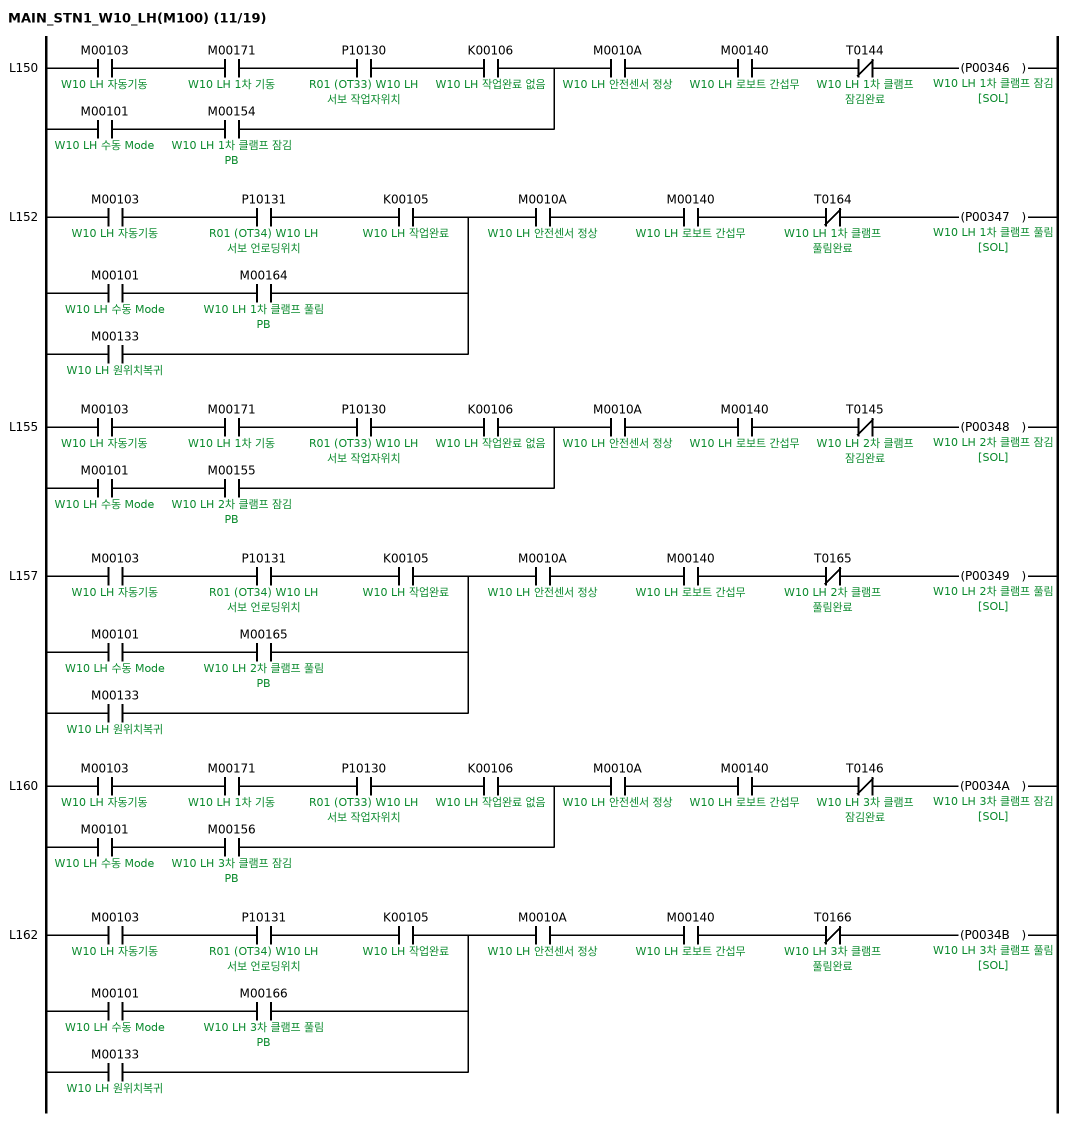
[picture p48: MAIN_STN1_W10_LH(M100) rungs L150-L162]
; L150
LOAD      M00103	// W10 LH 자동기동
AND       M00171	// W10 LH 1차 기동
AND       P10130	// R01 (OT33) W10 LH 서보 작업자위치
AND       K00106	// W10 LH 작업완료 없음
LOAD      M00101	// W10 LH 수동 Mode
AND       M00154	// W10 LH 1차 클램프 잠김 PB
OR LOAD
AND       M0010A	// W10 LH 안전센서 정상
AND       M00140	// W10 LH 로보트 간섭무
AND NOT   T0144	// W10 LH 1차 클램프 잠김완료
OUT       P00346	// W10 LH 1차 클램프 잠김 [SOL]
; L152
LOAD      M00103	// W10 LH 자동기동
AND       P10131	// R01 (OT34) W10 LH 서보 언로딩위치
AND       K00105	// W10 LH 작업완료
LOAD      M00101	// W10 LH 수동 Mode
AND       M00164	// W10 LH 1차 클램프 풀림 PB
OR LOAD
OR        M00133	// W10 LH 원위치복귀
AND       M0010A	// W10 LH 안전센서 정상
AND       M00140	// W10 LH 로보트 간섭무
AND NOT   T0164	// W10 LH 1차 클램프 풀림완료
OUT       P00347	// W10 LH 1차 클램프 풀림 [SOL]
; L155
LOAD      M00103	// W10 LH 자동기동
AND       M00171	// W10 LH 1차 기동
AND       P10130	// R01 (OT33) W10 LH 서보 작업자위치
AND       K00106	// W10 LH 작업완료 없음
LOAD      M00101	// W10 LH 수동 Mode
AND       M00155	// W10 LH 2차 클램프 잠김 PB
OR LOAD
AND       M0010A	// W10 LH 안전센서 정상
AND       M00140	// W10 LH 로보트 간섭무
AND NOT   T0145	// W10 LH 2차 클램프 잠김완료
OUT       P00348	// W10 LH 2차 클램프 잠김 [SOL]
; L157
LOAD      M00103	// W10 LH 자동기동
AND       P10131	// R01 (OT34) W10 LH 서보 언로딩위치
AND       K00105	// W10 LH 작업완료
LOAD      M00101	// W10 LH 수동 Mode
AND       M00165	// W10 LH 2차 클램프 풀림 PB
OR LOAD
OR        M00133	// W10 LH 원위치복귀
AND       M0010A	// W10 LH 안전센서 정상
AND       M00140	// W10 LH 로보트 간섭무
AND NOT   T0165	// W10 LH 2차 클램프 풀림완료
OUT       P00349	// W10 LH 2차 클램프 풀림 [SOL]
; L160
LOAD      M00103	// W10 LH 자동기동
AND       M00171	// W10 LH 1차 기동
AND       P10130	// R01 (OT33) W10 LH 서보 작업자위치
AND       K00106	// W10 LH 작업완료 없음
LOAD      M00101	// W10 LH 수동 Mode
AND       M00156	// W10 LH 3차 클램프 잠김 PB
OR LOAD
AND       M0010A	// W10 LH 안전센서 정상
AND       M00140	// W10 LH 로보트 간섭무
AND NOT   T0146	// W10 LH 3차 클램프 잠김완료
OUT       P0034A	// W10 LH 3차 클램프 잠김 [SOL]
; L162
LOAD      M00103	// W10 LH 자동기동
AND       P10131	// R01 (OT34) W10 LH 서보 언로딩위치
AND       K00105	// W10 LH 작업완료
LOAD      M00101	// W10 LH 수동 Mode
AND       M00166	// W10 LH 3차 클램프 풀림 PB
OR LOAD
OR        M00133	// W10 LH 원위치복귀
AND       M0010A	// W10 LH 안전센서 정상
AND       M00140	// W10 LH 로보트 간섭무
AND NOT   T0166	// W10 LH 3차 클램프 풀림완료
OUT       P0034B	// W10 LH 3차 클램프 풀림 [SOL]

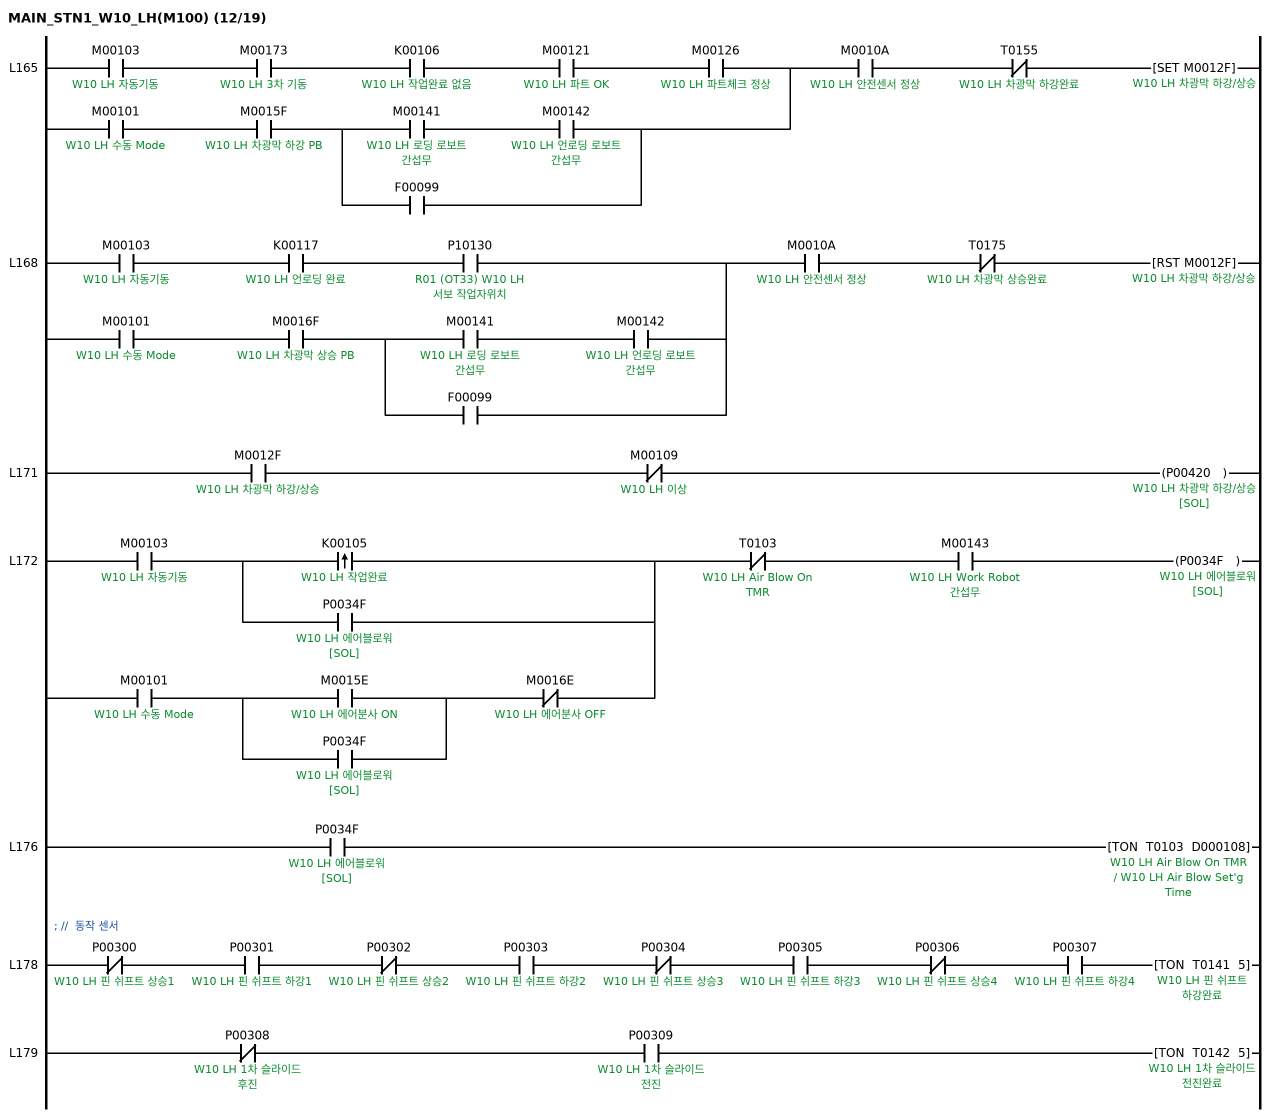
; L165
LOAD      M00103	// W10 LH 자동기동
AND       M00173	// W10 LH 3차 기동
AND       K00106	// W10 LH 작업완료 없음
AND       M00121	// W10 LH 파트 OK
AND       M00126	// W10 LH 파트체크 정상
LOAD      M00101	// W10 LH 수동 Mode
AND       M0015F	// W10 LH 차광막 하강 PB
LOAD      M00141	// W10 LH 로딩 로보트 간섭무
AND       M00142	// W10 LH 언로딩 로보트 간섭무
OR        F00099
AND LOAD
OR LOAD
AND       M0010A	// W10 LH 안전센서 정상
AND NOT   T0155	// W10 LH 차광막 하강완료
SET       M0012F	// W10 LH 차광막 하강/상승
; L168
LOAD      M00103	// W10 LH 자동기동
AND       K00117	// W10 LH 언로딩 완료
AND       P10130	// R01 (OT33) W10 LH 서보 작업자위치
LOAD      M00101	// W10 LH 수동 Mode
AND       M0016F	// W10 LH 차광막 상승 PB
LOAD      M00141	// W10 LH 로딩 로보트 간섭무
AND       M00142	// W10 LH 언로딩 로보트 간섭무
OR        F00099
AND LOAD
OR LOAD
AND       M0010A	// W10 LH 안전센서 정상
AND NOT   T0175	// W10 LH 차광막 상승완료
RST       M0012F	// W10 LH 차광막 하강/상승
; L171
LOAD      M0012F	// W10 LH 차광막 하강/상승
AND NOT   M00109	// W10 LH 이상
OUT       P00420	// W10 LH 차광막 하강/상승 [SOL]
; L172
LOAD      M00103	// W10 LH 자동기동
LOADP     K00105	// W10 LH 작업완료
OR        P0034F	// W10 LH 에어블로워 [SOL]
AND LOAD
LOAD      M00101	// W10 LH 수동 Mode
LOAD      M0015E	// W10 LH 에어분사 ON
OR        P0034F	// W10 LH 에어블로워 [SOL]
AND LOAD
AND NOT   M0016E	// W10 LH 에어분사 OFF
OR LOAD
AND NOT   T0103	// W10 LH Air Blow On TMR
AND       M00143	// W10 LH Work Robot 간섭무
OUT       P0034F	// W10 LH 에어블로워 [SOL]
; L176
LOAD      P0034F	// W10 LH 에어블로워 [SOL]
TON       T0103 D000108	// W10 LH Air Blow On TMR / W10 LH Air Blow Set'g Time
//   //  동작 센서
; L178
LOAD NOT  P00300	// W10 LH 핀 쉬프트 상승1
AND       P00301	// W10 LH 핀 쉬프트 하강1
AND NOT   P00302	// W10 LH 핀 쉬프트 상승2
AND       P00303	// W10 LH 핀 쉬프트 하강2
AND NOT   P00304	// W10 LH 핀 쉬프트 상승3
AND       P00305	// W10 LH 핀 쉬프트 하강3
AND NOT   P00306	// W10 LH 핀 쉬프트 상승4
AND       P00307	// W10 LH 핀 쉬프트 하강4
TON       T0141 5	// W10 LH 핀 쉬프트 하강완료
; L179
LOAD NOT  P00308	// W10 LH 1차 슬라이드 후진
AND       P00309	// W10 LH 1차 슬라이드 전진
TON       T0142 5	// W10 LH 1차 슬라이드 전진완료

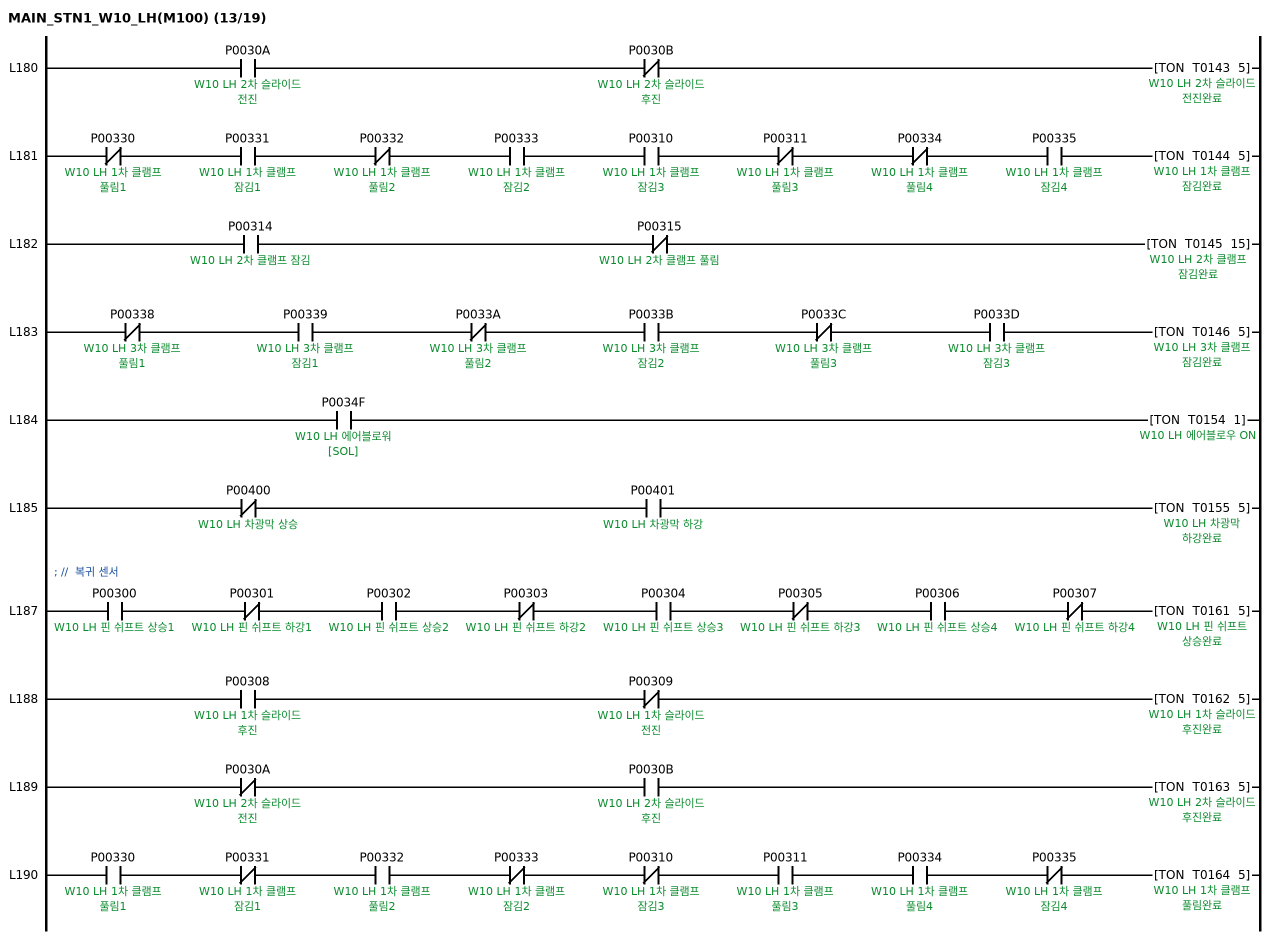
; L180
LOAD      P0030A	// W10 LH 2차 슬라이드 전진
AND NOT   P0030B	// W10 LH 2차 슬라이드 후진
TON       T0143 5	// W10 LH 2차 슬라이드 전진완료
; L181
LOAD NOT  P00330	// W10 LH 1차 클램프 풀림1
AND       P00331	// W10 LH 1차 클램프 잠김1
AND NOT   P00332	// W10 LH 1차 클램프 풀림2
AND       P00333	// W10 LH 1차 클램프 잠김2
AND       P00310	// W10 LH 1차 클램프 잠김3
AND NOT   P00311	// W10 LH 1차 클램프 풀림3
AND NOT   P00334	// W10 LH 1차 클램프 풀림4
AND       P00335	// W10 LH 1차 클램프 잠김4
TON       T0144 5	// W10 LH 1차 클램프 잠김완료
; L182
LOAD      P00314	// W10 LH 2차 클램프 잠김
AND NOT   P00315	// W10 LH 2차 클램프 풀림
TON       T0145 15	// W10 LH 2차 클램프 잠김완료
; L183
LOAD NOT  P00338	// W10 LH 3차 클램프 풀림1
AND       P00339	// W10 LH 3차 클램프 잠김1
AND NOT   P0033A	// W10 LH 3차 클램프 풀림2
AND       P0033B	// W10 LH 3차 클램프 잠김2
AND NOT   P0033C	// W10 LH 3차 클램프 풀림3
AND       P0033D	// W10 LH 3차 클램프 잠김3
TON       T0146 5	// W10 LH 3차 클램프 잠김완료
; L184
LOAD      P0034F	// W10 LH 에어블로워 [SOL]
TON       T0154 1	// W10 LH 에어블로우 ON
; L185
LOAD NOT  P00400	// W10 LH 차광막 상승
AND       P00401	// W10 LH 차광막 하강
TON       T0155 5	// W10 LH 차광막 하강완료
//   //  복귀 센서
; L187
LOAD      P00300	// W10 LH 핀 쉬프트 상승1
AND NOT   P00301	// W10 LH 핀 쉬프트 하강1
AND       P00302	// W10 LH 핀 쉬프트 상승2
AND NOT   P00303	// W10 LH 핀 쉬프트 하강2
AND       P00304	// W10 LH 핀 쉬프트 상승3
AND NOT   P00305	// W10 LH 핀 쉬프트 하강3
AND       P00306	// W10 LH 핀 쉬프트 상승4
AND NOT   P00307	// W10 LH 핀 쉬프트 하강4
TON       T0161 5	// W10 LH 핀 쉬프트 상승완료
; L188
LOAD      P00308	// W10 LH 1차 슬라이드 후진
AND NOT   P00309	// W10 LH 1차 슬라이드 전진
TON       T0162 5	// W10 LH 1차 슬라이드 후진완료
; L189
LOAD NOT  P0030A	// W10 LH 2차 슬라이드 전진
AND       P0030B	// W10 LH 2차 슬라이드 후진
TON       T0163 5	// W10 LH 2차 슬라이드 후진완료
; L190
LOAD      P00330	// W10 LH 1차 클램프 풀림1
AND NOT   P00331	// W10 LH 1차 클램프 잠김1
AND       P00332	// W10 LH 1차 클램프 풀림2
AND NOT   P00333	// W10 LH 1차 클램프 잠김2
AND NOT   P00310	// W10 LH 1차 클램프 잠김3
AND       P00311	// W10 LH 1차 클램프 풀림3
AND       P00334	// W10 LH 1차 클램프 풀림4
AND NOT   P00335	// W10 LH 1차 클램프 잠김4
TON       T0164 5	// W10 LH 1차 클램프 풀림완료

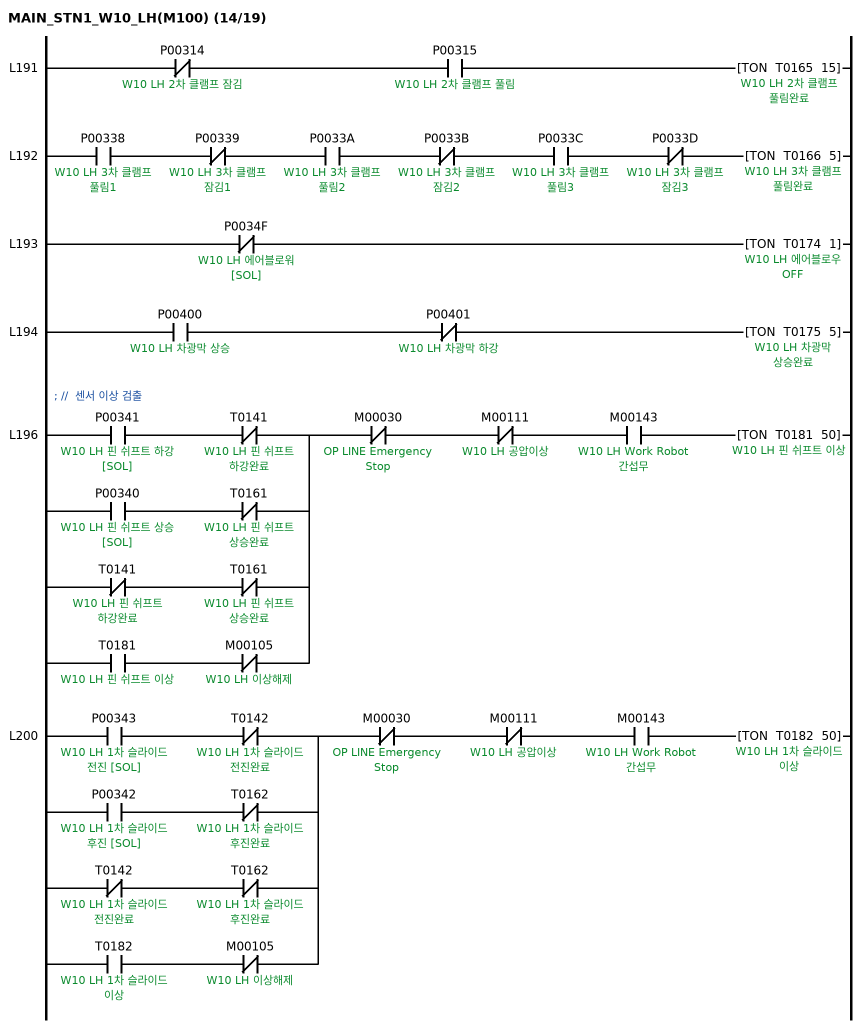
; L191
LOAD NOT  P00314	// W10 LH 2차 클램프 잠김
AND       P00315	// W10 LH 2차 클램프 풀림
TON       T0165 15	// W10 LH 2차 클램프 풀림완료
; L192
LOAD      P00338	// W10 LH 3차 클램프 풀림1
AND NOT   P00339	// W10 LH 3차 클램프 잠김1
AND       P0033A	// W10 LH 3차 클램프 풀림2
AND NOT   P0033B	// W10 LH 3차 클램프 잠김2
AND       P0033C	// W10 LH 3차 클램프 풀림3
AND NOT   P0033D	// W10 LH 3차 클램프 잠김3
TON       T0166 5	// W10 LH 3차 클램프 풀림완료
; L193
LOAD NOT  P0034F	// W10 LH 에어블로워 [SOL]
TON       T0174 1	// W10 LH 에어블로우 OFF
; L194
LOAD      P00400	// W10 LH 차광막 상승
AND NOT   P00401	// W10 LH 차광막 하강
TON       T0175 5	// W10 LH 차광막 상승완료
//     //  센서 이상 검출
; L196
LOAD      P00341	// W10 LH 핀 쉬프트 하강 [SOL]
AND NOT   T0141	// W10 LH 핀 쉬프트 하강완료
LOAD      P00340	// W10 LH 핀 쉬프트 상승 [SOL]
AND NOT   T0161	// W10 LH 핀 쉬프트 상승완료
OR LOAD
LOAD NOT  T0141	// W10 LH 핀 쉬프트 하강완료
AND NOT   T0161	// W10 LH 핀 쉬프트 상승완료
OR LOAD
LOAD      T0181	// W10 LH 핀 쉬프트 이상
AND NOT   M00105	// W10 LH 이상해제
OR LOAD
AND NOT   M00030	// OP LINE Emergency Stop
AND NOT   M00111	// W10 LH 공압이상
AND       M00143	// W10 LH Work Robot 간섭무
TON       T0181 50	// W10 LH 핀 쉬프트 이상
; L200
LOAD      P00343	// W10 LH 1차 슬라이드 전진 [SOL]
AND NOT   T0142	// W10 LH 1차 슬라이드 전진완료
LOAD      P00342	// W10 LH 1차 슬라이드 후진 [SOL]
AND NOT   T0162	// W10 LH 1차 슬라이드 후진완료
OR LOAD
LOAD NOT  T0142	// W10 LH 1차 슬라이드 전진완료
AND NOT   T0162	// W10 LH 1차 슬라이드 후진완료
OR LOAD
LOAD      T0182	// W10 LH 1차 슬라이드 이상
AND NOT   M00105	// W10 LH 이상해제
OR LOAD
AND NOT   M00030	// OP LINE Emergency Stop
AND NOT   M00111	// W10 LH 공압이상
AND       M00143	// W10 LH Work Robot 간섭무
TON       T0182 50	// W10 LH 1차 슬라이드 이상

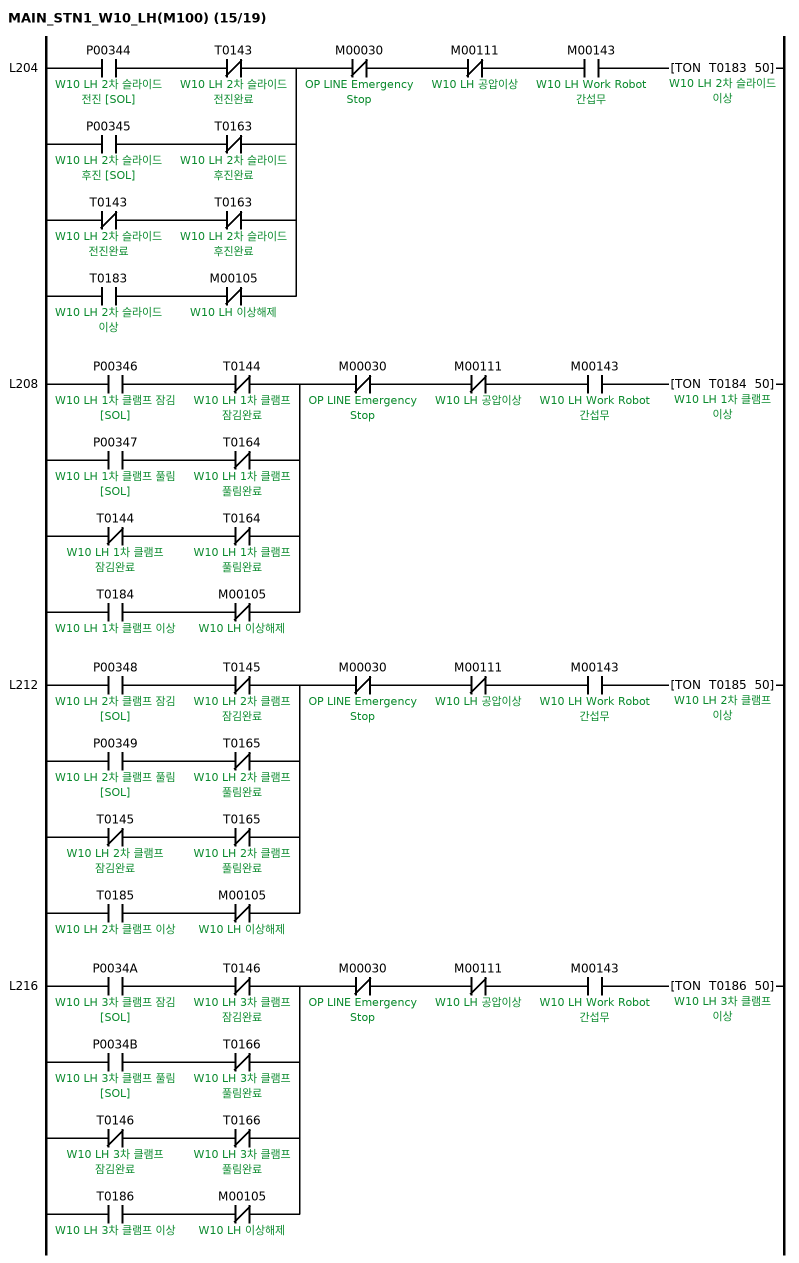
; L204
LOAD      P00344	// W10 LH 2차 슬라이드 전진 [SOL]
AND NOT   T0143	// W10 LH 2차 슬라이드 전진완료
LOAD      P00345	// W10 LH 2차 슬라이드 후진 [SOL]
AND NOT   T0163	// W10 LH 2차 슬라이드 후진완료
OR LOAD
LOAD NOT  T0143	// W10 LH 2차 슬라이드 전진완료
AND NOT   T0163	// W10 LH 2차 슬라이드 후진완료
OR LOAD
LOAD      T0183	// W10 LH 2차 슬라이드 이상
AND NOT   M00105	// W10 LH 이상해제
OR LOAD
AND NOT   M00030	// OP LINE Emergency Stop
AND NOT   M00111	// W10 LH 공압이상
AND       M00143	// W10 LH Work Robot 간섭무
TON       T0183 50	// W10 LH 2차 슬라이드 이상
; L208
LOAD      P00346	// W10 LH 1차 클램프 잠김 [SOL]
AND NOT   T0144	// W10 LH 1차 클램프 잠김완료
LOAD      P00347	// W10 LH 1차 클램프 풀림 [SOL]
AND NOT   T0164	// W10 LH 1차 클램프 풀림완료
OR LOAD
LOAD NOT  T0144	// W10 LH 1차 클램프 잠김완료
AND NOT   T0164	// W10 LH 1차 클램프 풀림완료
OR LOAD
LOAD      T0184	// W10 LH 1차 클램프 이상
AND NOT   M00105	// W10 LH 이상해제
OR LOAD
AND NOT   M00030	// OP LINE Emergency Stop
AND NOT   M00111	// W10 LH 공압이상
AND       M00143	// W10 LH Work Robot 간섭무
TON       T0184 50	// W10 LH 1차 클램프 이상
; L212
LOAD      P00348	// W10 LH 2차 클램프 잠김 [SOL]
AND NOT   T0145	// W10 LH 2차 클램프 잠김완료
LOAD      P00349	// W10 LH 2차 클램프 풀림 [SOL]
AND NOT   T0165	// W10 LH 2차 클램프 풀림완료
OR LOAD
LOAD NOT  T0145	// W10 LH 2차 클램프 잠김완료
AND NOT   T0165	// W10 LH 2차 클램프 풀림완료
OR LOAD
LOAD      T0185	// W10 LH 2차 클램프 이상
AND NOT   M00105	// W10 LH 이상해제
OR LOAD
AND NOT   M00030	// OP LINE Emergency Stop
AND NOT   M00111	// W10 LH 공압이상
AND       M00143	// W10 LH Work Robot 간섭무
TON       T0185 50	// W10 LH 2차 클램프 이상
; L216
LOAD      P0034A	// W10 LH 3차 클램프 잠김 [SOL]
AND NOT   T0146	// W10 LH 3차 클램프 잠김완료
LOAD      P0034B	// W10 LH 3차 클램프 풀림 [SOL]
AND NOT   T0166	// W10 LH 3차 클램프 풀림완료
OR LOAD
LOAD NOT  T0146	// W10 LH 3차 클램프 잠김완료
AND NOT   T0166	// W10 LH 3차 클램프 풀림완료
OR LOAD
LOAD      T0186	// W10 LH 3차 클램프 이상
AND NOT   M00105	// W10 LH 이상해제
OR LOAD
AND NOT   M00030	// OP LINE Emergency Stop
AND NOT   M00111	// W10 LH 공압이상
AND       M00143	// W10 LH Work Robot 간섭무
TON       T0186 50	// W10 LH 3차 클램프 이상

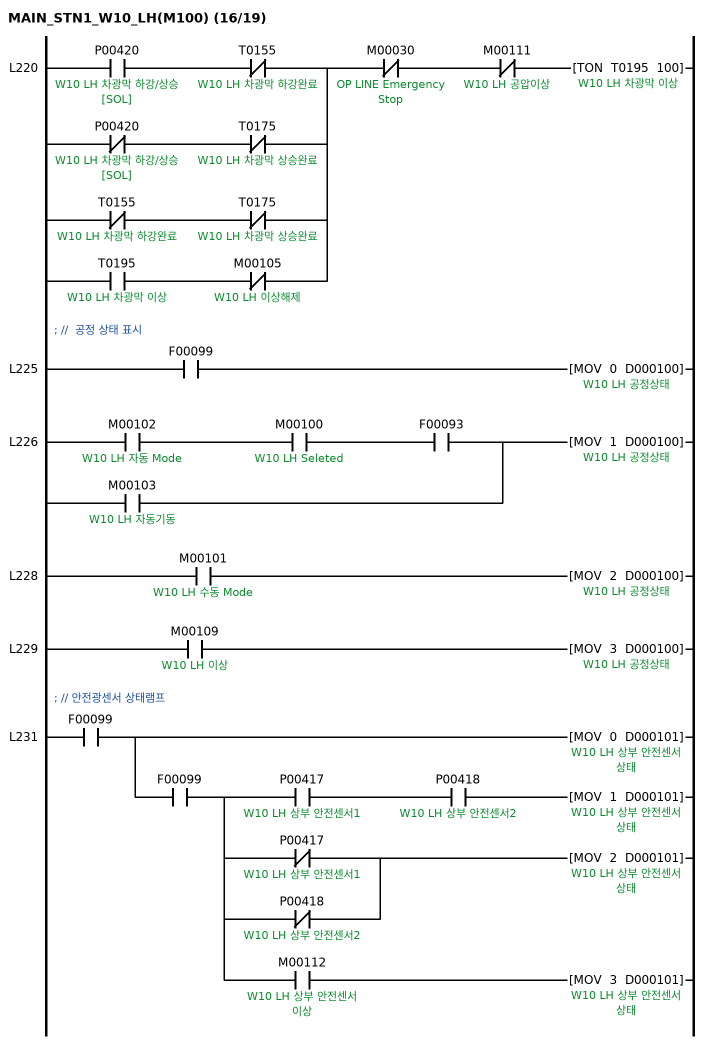
; L220
LOAD      P00420	// W10 LH 차광막 하강/상승 [SOL]
AND NOT   T0155	// W10 LH 차광막 하강완료
LOAD NOT  P00420	// W10 LH 차광막 하강/상승 [SOL]
AND NOT   T0175	// W10 LH 차광막 상승완료
OR LOAD
LOAD NOT  T0155	// W10 LH 차광막 하강완료
AND NOT   T0175	// W10 LH 차광막 상승완료
OR LOAD
LOAD      T0195	// W10 LH 차광막 이상
AND NOT   M00105	// W10 LH 이상해제
OR LOAD
AND NOT   M00030	// OP LINE Emergency Stop
AND NOT   M00111	// W10 LH 공압이상
TON       T0195 100	// W10 LH 차광막 이상
//   //  공정 상태 표시
; L225
LOAD      F00099
MOV       0 D000100	// W10 LH 공정상태
; L226
LOAD      M00102	// W10 LH 자동 Mode
AND       M00100	// W10 LH Seleted
AND       F00093
OR        M00103	// W10 LH 자동기동
MOV       1 D000100	// W10 LH 공정상태
; L228
LOAD      M00101	// W10 LH 수동 Mode
MOV       2 D000100	// W10 LH 공정상태
; L229
LOAD      M00109	// W10 LH 이상
MOV       3 D000100	// W10 LH 공정상태
//   // 안전광센서 상태램프
; L231
LOAD      F00099
MOV       0 D000101	// W10 LH 상부 안전센서 상태
AND       F00099
MPUSH
AND       P00417	// W10 LH 상부 안전센서1
AND       P00418	// W10 LH 상부 안전센서2
MOV       1 D000101	// W10 LH 상부 안전센서 상태
MLOAD
LOAD NOT  P00417	// W10 LH 상부 안전센서1
OR NOT    P00418	// W10 LH 상부 안전센서2
AND LOAD
MOV       2 D000101	// W10 LH 상부 안전센서 상태
MPOP
AND       M00112	// W10 LH 상부 안전센서 이상
MOV       3 D000101	// W10 LH 상부 안전센서 상태

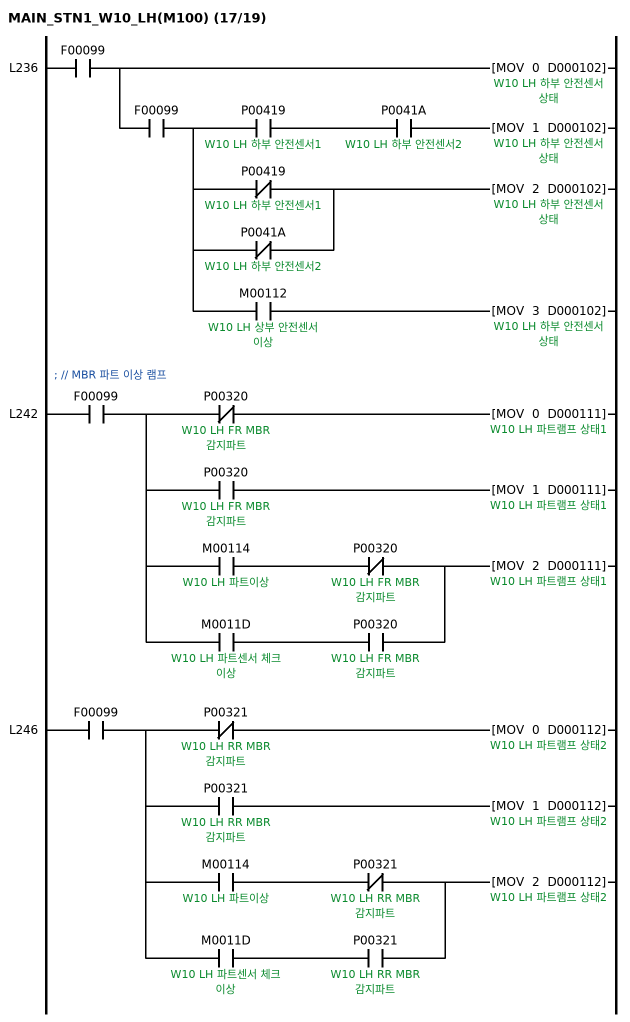
; L236
LOAD      F00099
MOV       0 D000102	// W10 LH 하부 안전센서 상태
AND       F00099
MPUSH
AND       P00419	// W10 LH 하부 안전센서1
AND       P0041A	// W10 LH 하부 안전센서2
MOV       1 D000102	// W10 LH 하부 안전센서 상태
MLOAD
LOAD NOT  P00419	// W10 LH 하부 안전센서1
OR NOT    P0041A	// W10 LH 하부 안전센서2
AND LOAD
MOV       2 D000102	// W10 LH 하부 안전센서 상태
MPOP
AND       M00112	// W10 LH 상부 안전센서 이상
MOV       3 D000102	// W10 LH 하부 안전센서 상태
//   // MBR 파트 이상 램프
; L242
LOAD      F00099
MPUSH
AND NOT   P00320	// W10 LH FR MBR 감지파트
MOV       0 D000111	// W10 LH 파트램프 상태1
MLOAD
AND       P00320	// W10 LH FR MBR 감지파트
MOV       1 D000111	// W10 LH 파트램프 상태1
MPOP
LOAD      M00114	// W10 LH 파트이상
AND NOT   P00320	// W10 LH FR MBR 감지파트
LOAD      M0011D	// W10 LH 파트센서 체크 이상
AND       P00320	// W10 LH FR MBR 감지파트
OR LOAD
AND LOAD
MOV       2 D000111	// W10 LH 파트램프 상태1
; L246
LOAD      F00099
MPUSH
AND NOT   P00321	// W10 LH RR MBR 감지파트
MOV       0 D000112	// W10 LH 파트램프 상태2
MLOAD
AND       P00321	// W10 LH RR MBR 감지파트
MOV       1 D000112	// W10 LH 파트램프 상태2
MPOP
LOAD      M00114	// W10 LH 파트이상
AND NOT   P00321	// W10 LH RR MBR 감지파트
LOAD      M0011D	// W10 LH 파트센서 체크 이상
AND       P00321	// W10 LH RR MBR 감지파트
OR LOAD
AND LOAD
MOV       2 D000112	// W10 LH 파트램프 상태2

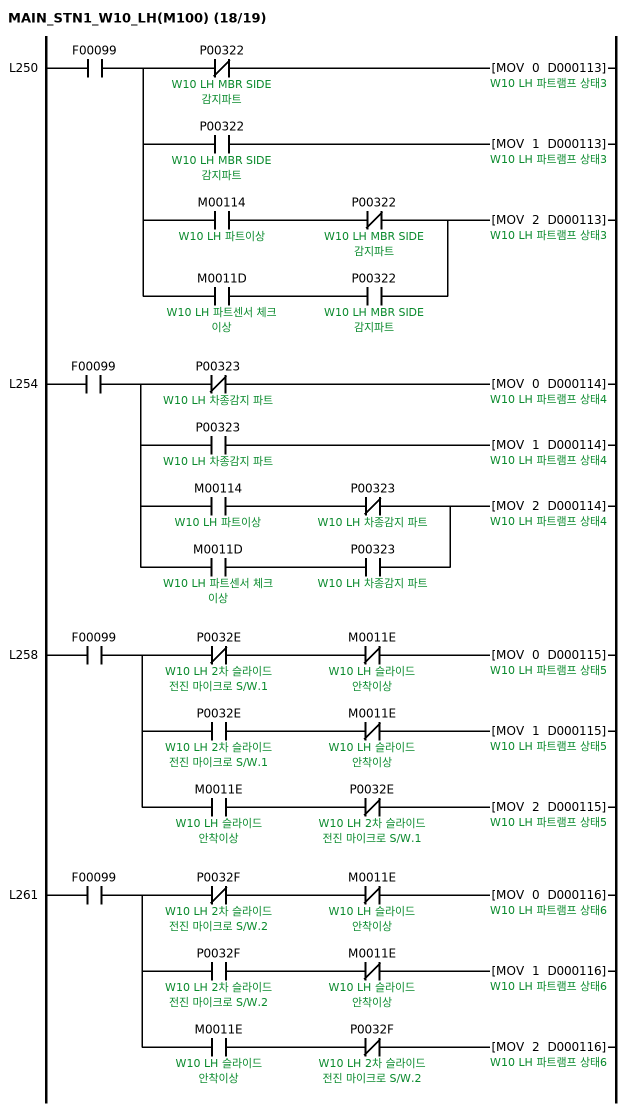
; L250
LOAD      F00099
MPUSH
AND NOT   P00322	// W10 LH MBR SIDE 감지파트
MOV       0 D000113	// W10 LH 파트램프 상태3
MLOAD
AND       P00322	// W10 LH MBR SIDE 감지파트
MOV       1 D000113	// W10 LH 파트램프 상태3
MPOP
LOAD      M00114	// W10 LH 파트이상
AND NOT   P00322	// W10 LH MBR SIDE 감지파트
LOAD      M0011D	// W10 LH 파트센서 체크 이상
AND       P00322	// W10 LH MBR SIDE 감지파트
OR LOAD
AND LOAD
MOV       2 D000113	// W10 LH 파트램프 상태3
; L254
LOAD      F00099
MPUSH
AND NOT   P00323	// W10 LH 차종감지 파트
MOV       0 D000114	// W10 LH 파트램프 상태4
MLOAD
AND       P00323	// W10 LH 차종감지 파트
MOV       1 D000114	// W10 LH 파트램프 상태4
MPOP
LOAD      M00114	// W10 LH 파트이상
AND NOT   P00323	// W10 LH 차종감지 파트
LOAD      M0011D	// W10 LH 파트센서 체크 이상
AND       P00323	// W10 LH 차종감지 파트
OR LOAD
AND LOAD
MOV       2 D000114	// W10 LH 파트램프 상태4
; L258
LOAD      F00099
MPUSH
AND NOT   P0032E	// W10 LH 2차 슬라이드 전진 마이크로 S/W.1
AND NOT   M0011E	// W10 LH 슬라이드 안착이상
MOV       0 D000115	// W10 LH 파트램프 상태5
MLOAD
AND       P0032E	// W10 LH 2차 슬라이드 전진 마이크로 S/W.1
AND NOT   M0011E	// W10 LH 슬라이드 안착이상
MOV       1 D000115	// W10 LH 파트램프 상태5
MPOP
AND       M0011E	// W10 LH 슬라이드 안착이상
AND NOT   P0032E	// W10 LH 2차 슬라이드 전진 마이크로 S/W.1
MOV       2 D000115	// W10 LH 파트램프 상태5
; L261
LOAD      F00099
MPUSH
AND NOT   P0032F	// W10 LH 2차 슬라이드 전진 마이크로 S/W.2
AND NOT   M0011E	// W10 LH 슬라이드 안착이상
MOV       0 D000116	// W10 LH 파트램프 상태6
MLOAD
AND       P0032F	// W10 LH 2차 슬라이드 전진 마이크로 S/W.2
AND NOT   M0011E	// W10 LH 슬라이드 안착이상
MOV       1 D000116	// W10 LH 파트램프 상태6
MPOP
AND       M0011E	// W10 LH 슬라이드 안착이상
AND NOT   P0032F	// W10 LH 2차 슬라이드 전진 마이크로 S/W.2
MOV       2 D000116	// W10 LH 파트램프 상태6

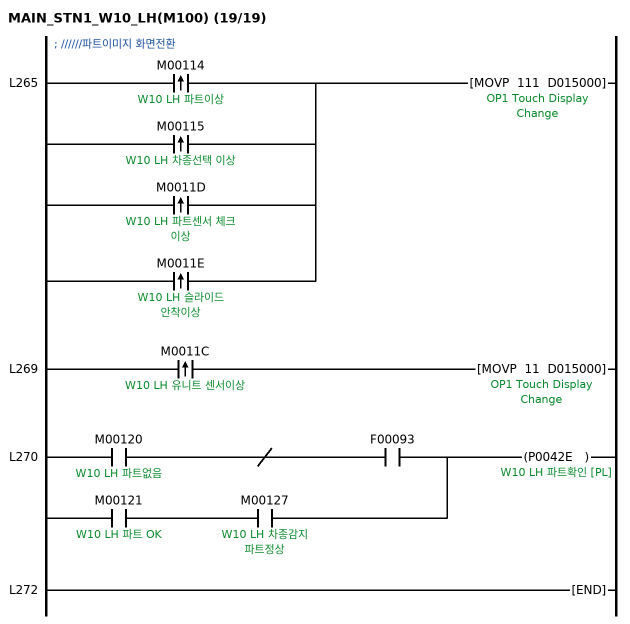
// //////파트이미지 화면전환
; L265
LOADP     M00114	// W10 LH 파트이상
ORP       M00115	// W10 LH 차종선택 이상
ORP       M0011D	// W10 LH 파트센서 체크 이상
ORP       M0011E	// W10 LH 슬라이드 안착이상
MOVP      111 D015000	// OP1 Touch Display Change
; L269
LOADP     M0011C	// W10 LH 유니트 센서이상
MOVP      11 D015000	// OP1 Touch Display Change
; L270
LOAD      M00120	// W10 LH 파트없음
NOT
AND       F00093
LOAD      M00121	// W10 LH 파트 OK
AND       M00127	// W10 LH 차종감지 파트정상
OR LOAD
OUT       P0042E	// W10 LH 파트확인 [PL]
; L272
END

PROGRAM MAIN_STN2_W10_RH(M200) (task: 스캔 프로그램)

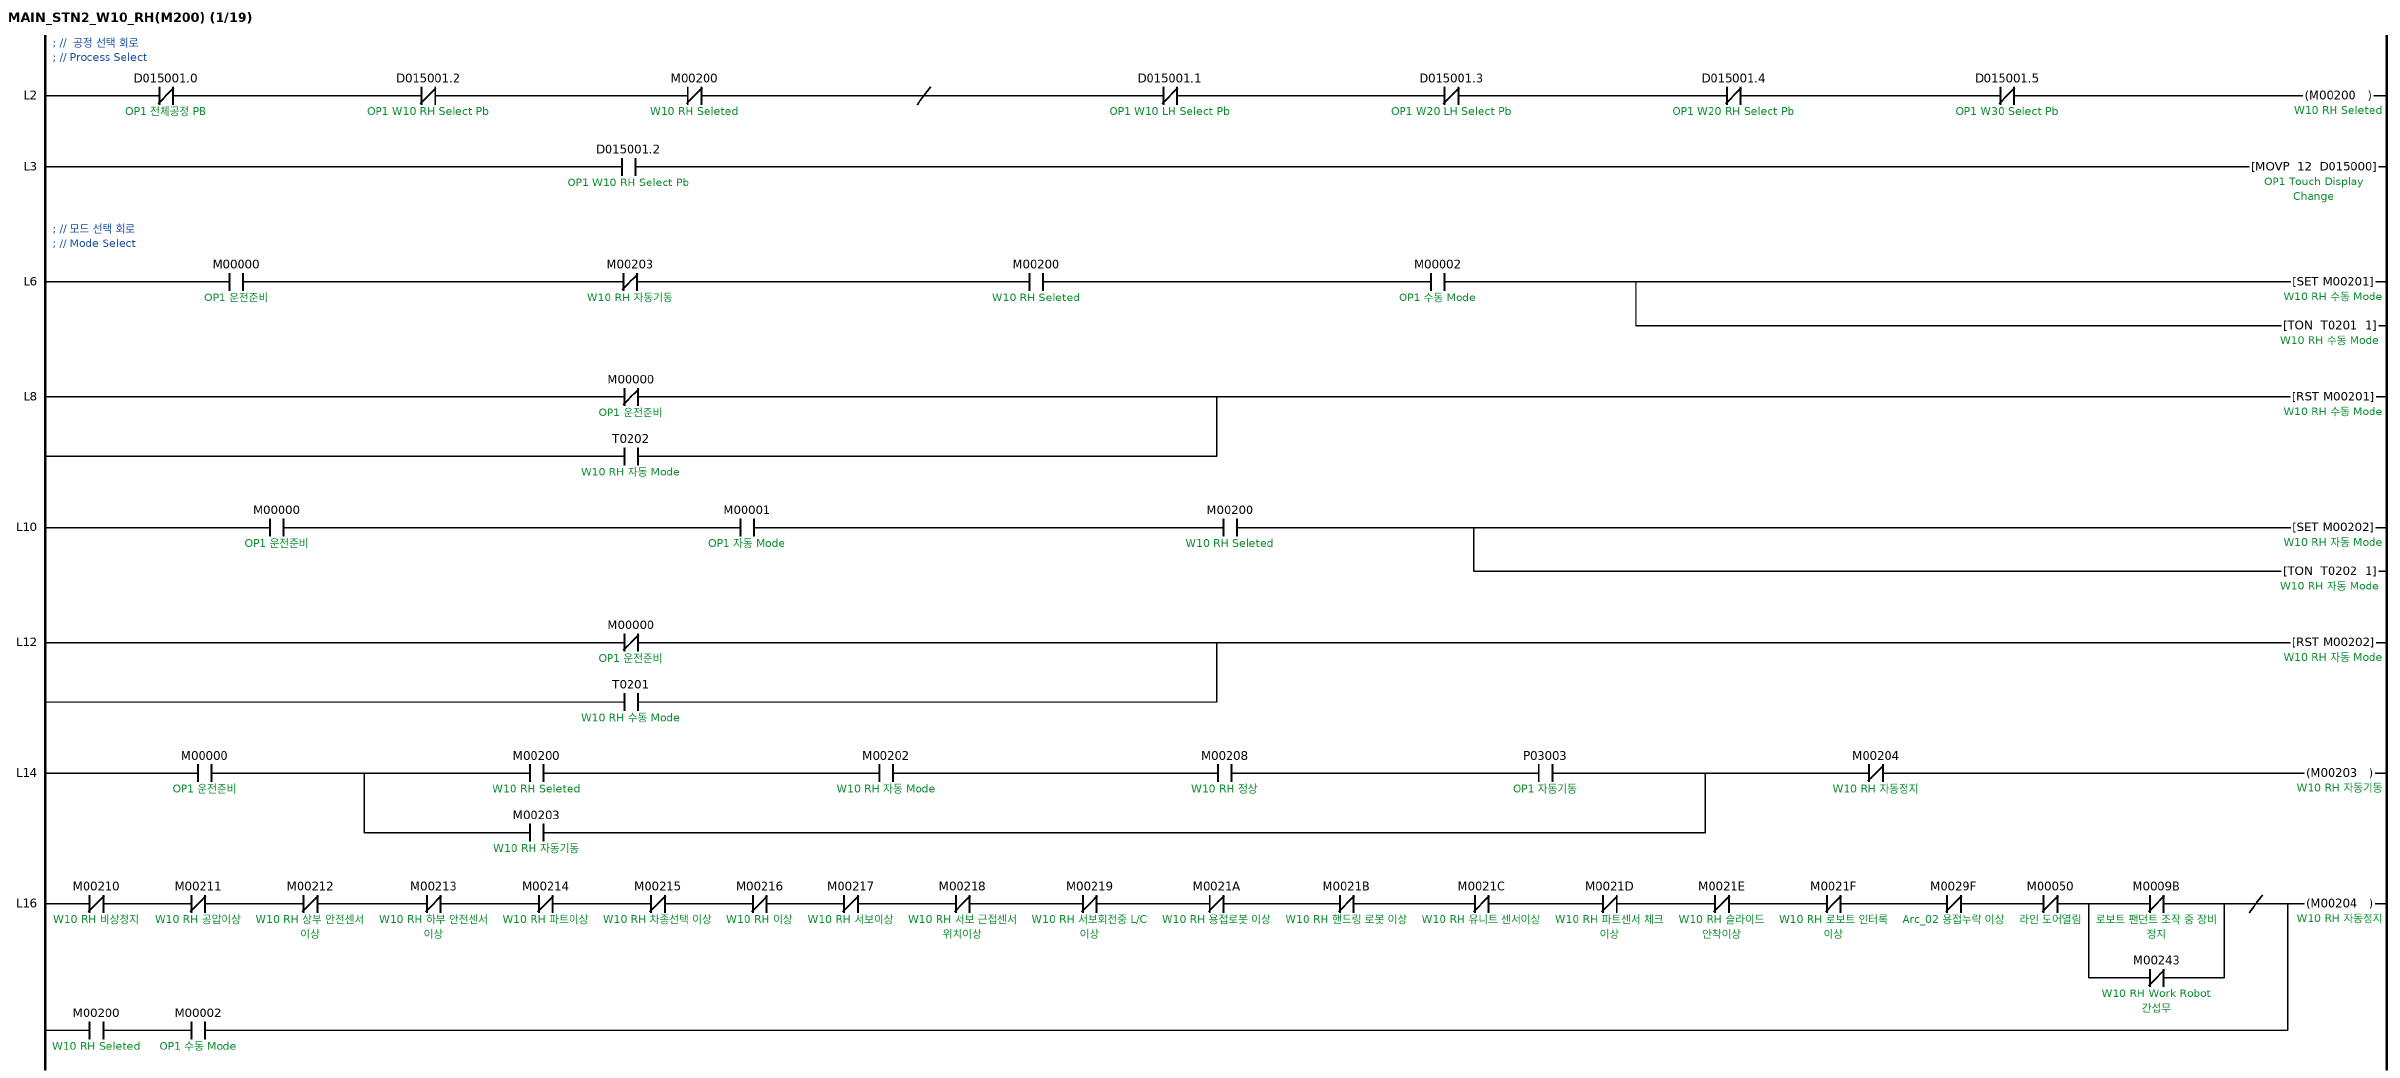
//   //  공정 선택 회로
//   // Process Select
; L2
LOAD NOT  D015001.0	// OP1 전체공정 PB
AND NOT   D015001.2	// OP1 W10 RH Select Pb
AND NOT   M00200	// W10 RH Seleted
NOT
AND NOT   D015001.1	// OP1 W10 LH Select Pb
AND NOT   D015001.3	// OP1 W20 LH Select Pb
AND NOT   D015001.4	// OP1 W20 RH Select Pb
AND NOT   D015001.5	// OP1 W30 Select Pb
OUT       M00200	// W10 RH Seleted
; L3
LOAD      D015001.2	// OP1 W10 RH Select Pb
MOVP      12 D015000	// OP1 Touch Display Change
// // 모드 선택 회로
//   // Mode Select
; L6
LOAD      M00000	// OP1 운전준비
AND NOT   M00203	// W10 RH 자동기동
AND       M00200	// W10 RH Seleted
AND       M00002	// OP1 수동 Mode
SET       M00201	// W10 RH 수동 Mode
TON       T0201 1	// W10 RH 수동 Mode
; L8
LOAD NOT  M00000	// OP1 운전준비
OR        T0202	// W10 RH 자동 Mode
RST       M00201	// W10 RH 수동 Mode
; L10
LOAD      M00000	// OP1 운전준비
AND       M00001	// OP1 자동 Mode
AND       M00200	// W10 RH Seleted
SET       M00202	// W10 RH 자동 Mode
TON       T0202 1	// W10 RH 자동 Mode
; L12
LOAD NOT  M00000	// OP1 운전준비
OR        T0201	// W10 RH 수동 Mode
RST       M00202	// W10 RH 자동 Mode
; L14
LOAD      M00000	// OP1 운전준비
LOAD      M00200	// W10 RH Seleted
AND       M00202	// W10 RH 자동 Mode
AND       M00208	// W10 RH 정상
AND       P03003	// OP1 자동기동
OR        M00203	// W10 RH 자동기동
AND LOAD
AND NOT   M00204	// W10 RH 자동정지
OUT       M00203	// W10 RH 자동기동
; L16
LOAD NOT  M00210	// W10 RH 비상정지
AND NOT   M00211	// W10 RH 공압이상
AND NOT   M00212	// W10 RH 상부 안전센서 이상
AND NOT   M00213	// W10 RH 하부 안전센서 이상
AND NOT   M00214	// W10 RH 파트이상
AND NOT   M00215	// W10 RH 차종선택 이상
AND NOT   M00216	// W10 RH 이상
AND NOT   M00217	// W10 RH 서보이상
AND NOT   M00218	// W10 RH 서보 근접센서 위치이상
AND NOT   M00219	// W10 RH 서보회전중 L/C 이상
AND NOT   M0021A	// W10 RH 용접로봇 이상
AND NOT   M0021B	// W10 RH 핸드링 로봇 이상
AND NOT   M0021C	// W10 RH 유니트 센서이상
AND NOT   M0021D	// W10 RH 파트센서 체크 이상
AND NOT   M0021E	// W10 RH 슬라이드 안착이상
AND NOT   M0021F	// W10 RH 로보트 인터록 이상
AND NOT   M0029F	// Arc_02 용접누락 이상
AND NOT   M00050	// 라인 도어열림
LOAD NOT  M0009B	// 로보트 팬던트 조작 중 장비 정지
OR NOT    M00243	// W10 RH Work Robot 간섭무
AND LOAD
NOT
LOAD      M00200	// W10 RH Seleted
AND       M00002	// OP1 수동 Mode
OR LOAD
OUT       M00204	// W10 RH 자동정지

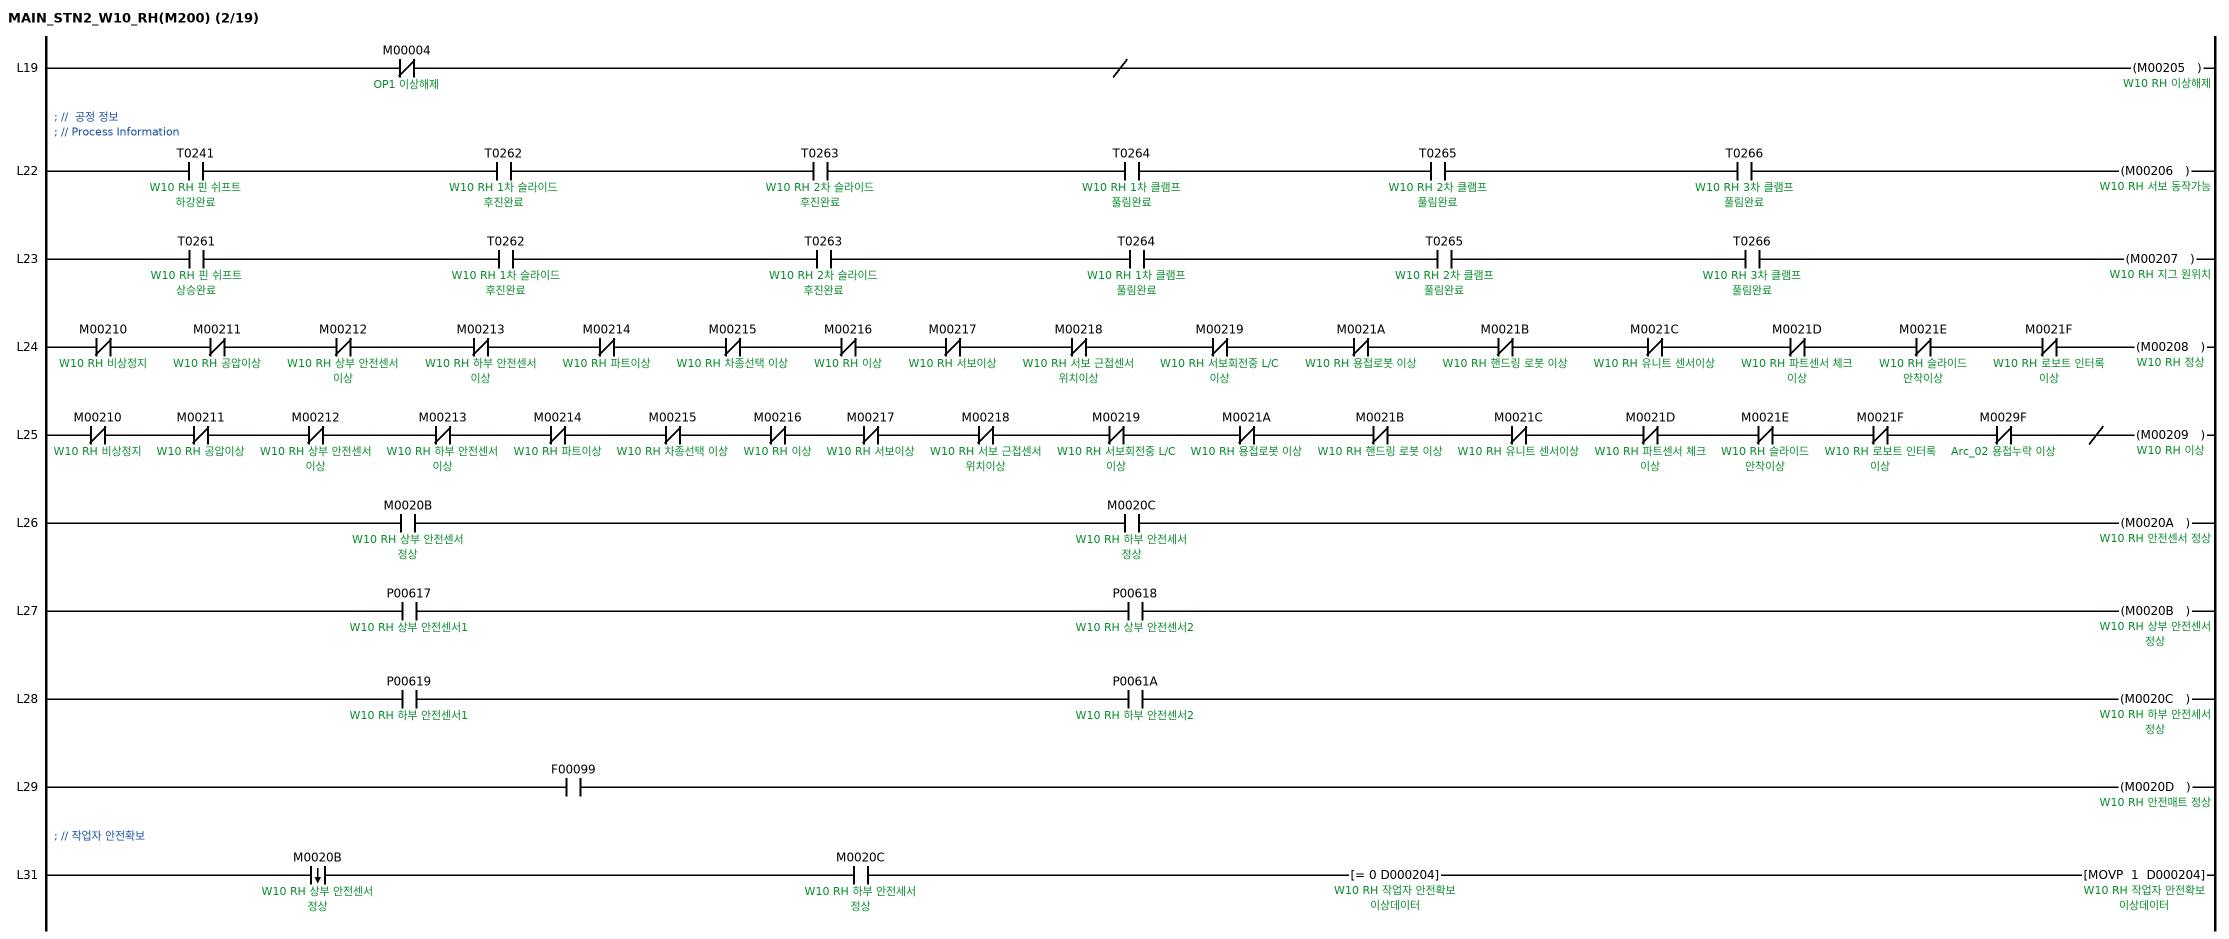
; L19
LOAD NOT  M00004	// OP1 이상해제
NOT
OUT       M00205	// W10 RH 이상해제
//   //  공정 정보
//   // Process Information
; L22
LOAD      T0241	// W10 RH 핀 쉬프트 하강완료
AND       T0262	// W10 RH 1차 슬라이드 후진완료
AND       T0263	// W10 RH 2차 슬라이드 후진완료
AND       T0264	// W10 RH 1차 클램프 풀림완료
AND       T0265	// W10 RH 2차 클램프 풀림완료
AND       T0266	// W10 RH 3차 클램프 풀림완료
OUT       M00206	// W10 RH 서보 동작가능
; L23
LOAD      T0261	// W10 RH 핀 쉬프트 상승완료
AND       T0262	// W10 RH 1차 슬라이드 후진완료
AND       T0263	// W10 RH 2차 슬라이드 후진완료
AND       T0264	// W10 RH 1차 클램프 풀림완료
AND       T0265	// W10 RH 2차 클램프 풀림완료
AND       T0266	// W10 RH 3차 클램프 풀림완료
OUT       M00207	// W10 RH 지그 원위치
; L24
LOAD NOT  M00210	// W10 RH 비상정지
AND NOT   M00211	// W10 RH 공압이상
AND NOT   M00212	// W10 RH 상부 안전센서 이상
AND NOT   M00213	// W10 RH 하부 안전센서 이상
AND NOT   M00214	// W10 RH 파트이상
AND NOT   M00215	// W10 RH 차종선택 이상
AND NOT   M00216	// W10 RH 이상
AND NOT   M00217	// W10 RH 서보이상
AND NOT   M00218	// W10 RH 서보 근접센서 위치이상
AND NOT   M00219	// W10 RH 서보회전중 L/C 이상
AND NOT   M0021A	// W10 RH 용접로봇 이상
AND NOT   M0021B	// W10 RH 핸드링 로봇 이상
AND NOT   M0021C	// W10 RH 유니트 센서이상
AND NOT   M0021D	// W10 RH 파트센서 체크 이상
AND NOT   M0021E	// W10 RH 슬라이드 안착이상
AND NOT   M0021F	// W10 RH 로보트 인터록 이상
OUT       M00208	// W10 RH 정상
; L25
LOAD NOT  M00210	// W10 RH 비상정지
AND NOT   M00211	// W10 RH 공압이상
AND NOT   M00212	// W10 RH 상부 안전센서 이상
AND NOT   M00213	// W10 RH 하부 안전센서 이상
AND NOT   M00214	// W10 RH 파트이상
AND NOT   M00215	// W10 RH 차종선택 이상
AND NOT   M00216	// W10 RH 이상
AND NOT   M00217	// W10 RH 서보이상
AND NOT   M00218	// W10 RH 서보 근접센서 위치이상
AND NOT   M00219	// W10 RH 서보회전중 L/C 이상
AND NOT   M0021A	// W10 RH 용접로봇 이상
AND NOT   M0021B	// W10 RH 핸드링 로봇 이상
AND NOT   M0021C	// W10 RH 유니트 센서이상
AND NOT   M0021D	// W10 RH 파트센서 체크 이상
AND NOT   M0021E	// W10 RH 슬라이드 안착이상
AND NOT   M0021F	// W10 RH 로보트 인터록 이상
AND NOT   M0029F	// Arc_02 용접누락 이상
NOT
OUT       M00209	// W10 RH 이상
; L26
LOAD      M0020B	// W10 RH 상부 안전센서 정상
AND       M0020C	// W10 RH 하부 안전세서 정상
OUT       M0020A	// W10 RH 안전센서 정상
; L27
LOAD      P00617	// W10 RH 상부 안전센서1
AND       P00618	// W10 RH 상부 안전센서2
OUT       M0020B	// W10 RH 상부 안전센서 정상
; L28
LOAD      P00619	// W10 RH 하부 안전센서1
AND       P0061A	// W10 RH 하부 안전센서2
OUT       M0020C	// W10 RH 하부 안전세서 정상
; L29
LOAD      F00099
OUT       M0020D	// W10 RH 안전매트 정상
//    // 작업자 안전확보
; L31
LOADN     M0020B	// W10 RH 상부 안전센서 정상
AND       M0020C	// W10 RH 하부 안전세서 정상
AND=      0 D000204	// W10 RH 작업자 안전확보 이상데이터
MOVP      1 D000204	// W10 RH 작업자 안전확보 이상데이터

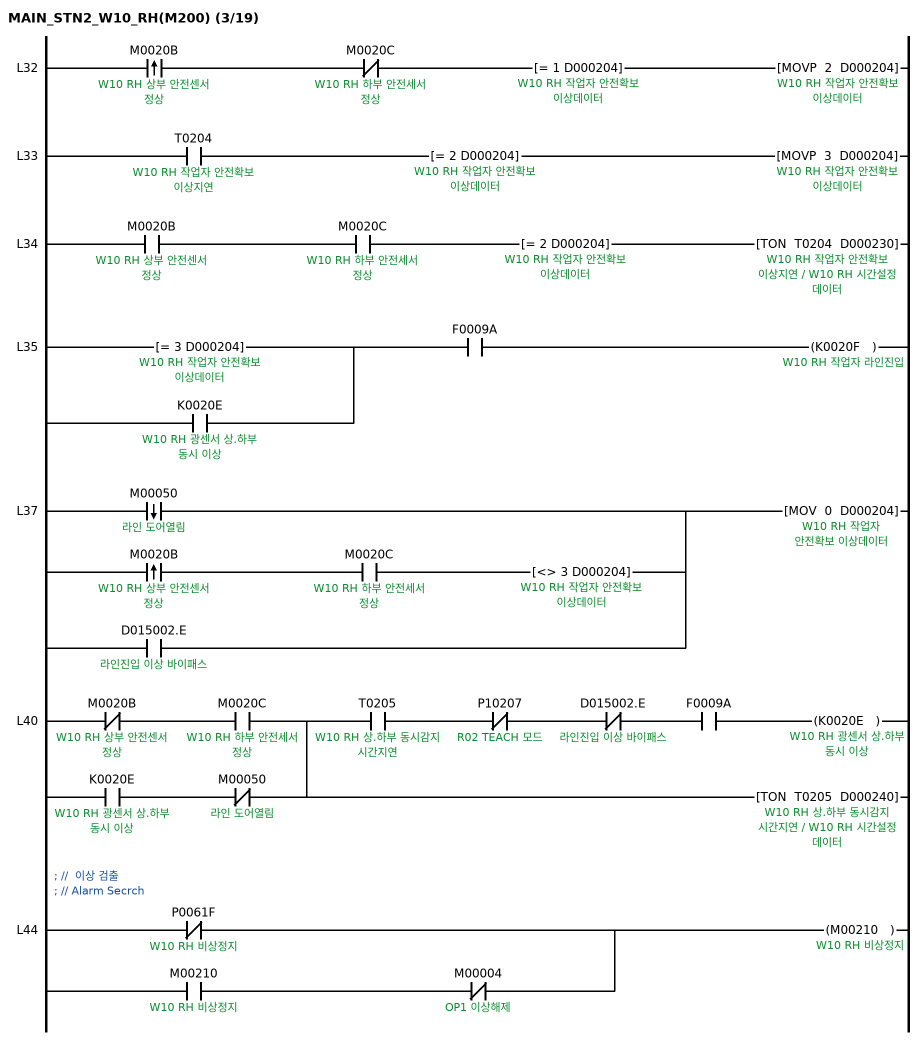
; L32
LOADP     M0020B	// W10 RH 상부 안전센서 정상
AND NOT   M0020C	// W10 RH 하부 안전세서 정상
AND=      1 D000204	// W10 RH 작업자 안전확보 이상데이터
MOVP      2 D000204	// W10 RH 작업자 안전확보 이상데이터
; L33
LOAD      T0204	// W10 RH 작업자 안전확보 이상지연
AND=      2 D000204	// W10 RH 작업자 안전확보 이상데이터
MOVP      3 D000204	// W10 RH 작업자 안전확보 이상데이터
; L34
LOAD      M0020B	// W10 RH 상부 안전센서 정상
AND       M0020C	// W10 RH 하부 안전세서 정상
AND=      2 D000204	// W10 RH 작업자 안전확보 이상데이터
TON       T0204 D000230	// W10 RH 작업자 안전확보 이상지연 / W10 RH 시간설정 데이터
; L35
LOAD=     3 D000204	// W10 RH 작업자 안전확보 이상데이터
OR        K0020E	// W10 RH 광센서 상.하부 동시 이상
AND       F0009A
OUT       K0020F	// W10 RH 작업자 라인진입
; L37
LOADN     M00050	// 라인 도어열림
LOADP     M0020B	// W10 RH 상부 안전센서 정상
AND       M0020C	// W10 RH 하부 안전세서 정상
AND<>     3 D000204	// W10 RH 작업자 안전확보 이상데이터
OR LOAD
OR        D015002.E	// 라인진입 이상 바이패스
MOV       0 D000204	// W10 RH 작업자 안전확보 이상데이터
; L40
LOAD NOT  M0020B	// W10 RH 상부 안전센서 정상
AND       M0020C	// W10 RH 하부 안전세서 정상
LOAD      K0020E	// W10 RH 광센서 상.하부 동시 이상
AND NOT   M00050	// 라인 도어열림
OR LOAD
MPUSH
AND       T0205	// W10 RH 상.하부 동시감지 시간지연
AND NOT   P10207	// R02 TEACH 모드
AND NOT   D015002.E	// 라인진입 이상 바이패스
AND       F0009A
OUT       K0020E	// W10 RH 광센서 상.하부 동시 이상
MPOP
TON       T0205 D000240	// W10 RH 상.하부 동시감지 시간지연 / W10 RH 시간설정 데이터
//   //  이상 검출
//   // Alarm Secrch
; L44
LOAD NOT  P0061F	// W10 RH 비상정지
LOAD      M00210	// W10 RH 비상정지
AND NOT   M00004	// OP1 이상해제
OR LOAD
OUT       M00210	// W10 RH 비상정지

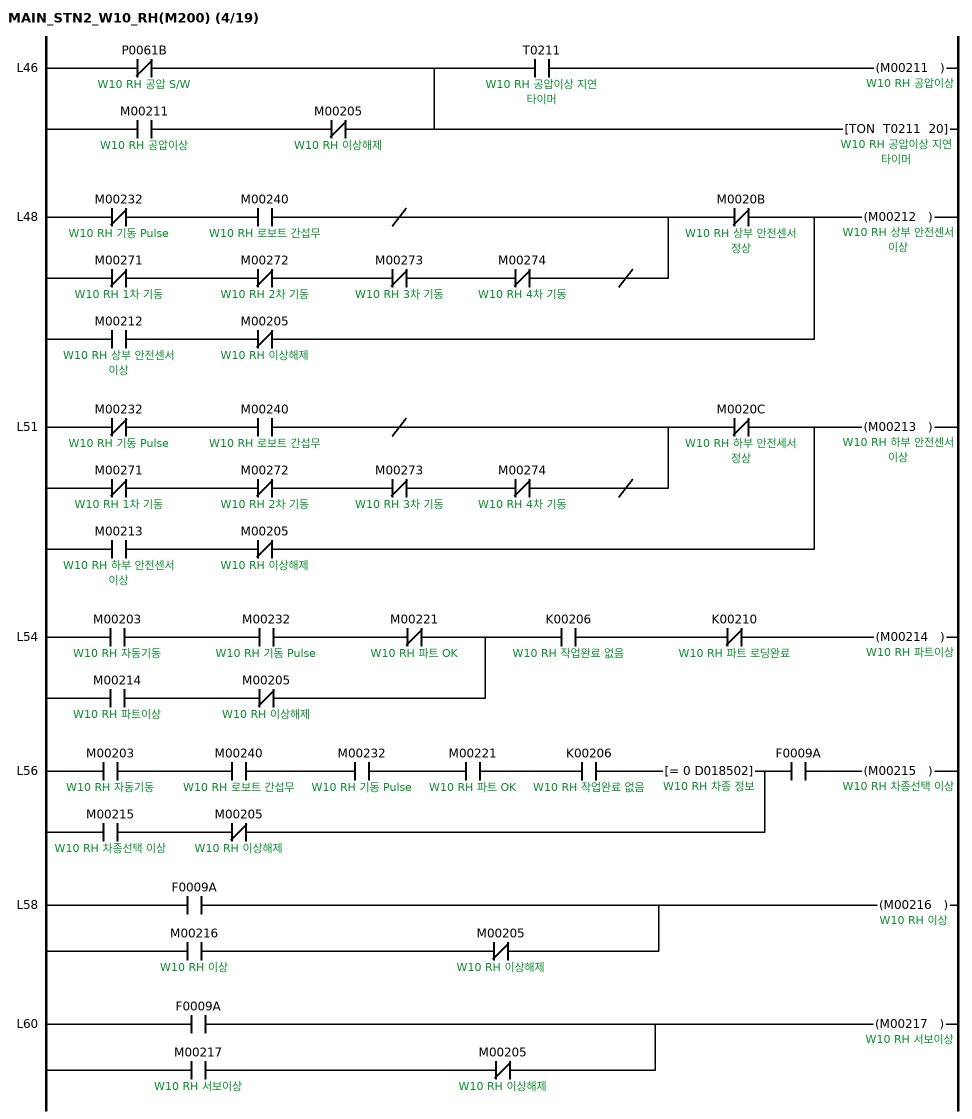
; L46
LOAD NOT  P0061B	// W10 RH 공압 S/W
LOAD      M00211	// W10 RH 공압이상
AND NOT   M00205	// W10 RH 이상해제
OR LOAD
MPUSH
AND       T0211	// W10 RH 공압이상 지연 타이머
OUT       M00211	// W10 RH 공압이상
MPOP
TON       T0211 20	// W10 RH 공압이상 지연 타이머
; L48
LOAD NOT  M00232	// W10 RH 기동 Pulse
AND       M00240	// W10 RH 로보트 간섭무
NOT
LOAD NOT  M00271	// W10 RH 1차 기동
AND NOT   M00272	// W10 RH 2차 기동
AND NOT   M00273	// W10 RH 3차 기동
AND NOT   M00274	// W10 RH 4차 기동
NOT
OR LOAD
AND NOT   M0020B	// W10 RH 상부 안전센서 정상
LOAD      M00212	// W10 RH 상부 안전센서 이상
AND NOT   M00205	// W10 RH 이상해제
OR LOAD
OUT       M00212	// W10 RH 상부 안전센서 이상
; L51
LOAD NOT  M00232	// W10 RH 기동 Pulse
AND       M00240	// W10 RH 로보트 간섭무
NOT
LOAD NOT  M00271	// W10 RH 1차 기동
AND NOT   M00272	// W10 RH 2차 기동
AND NOT   M00273	// W10 RH 3차 기동
AND NOT   M00274	// W10 RH 4차 기동
NOT
OR LOAD
AND NOT   M0020C	// W10 RH 하부 안전세서 정상
LOAD      M00213	// W10 RH 하부 안전센서 이상
AND NOT   M00205	// W10 RH 이상해제
OR LOAD
OUT       M00213	// W10 RH 하부 안전센서 이상
; L54
LOAD      M00203	// W10 RH 자동기동
AND       M00232	// W10 RH 기동 Pulse
AND NOT   M00221	// W10 RH 파트 OK
LOAD      M00214	// W10 RH 파트이상
AND NOT   M00205	// W10 RH 이상해제
OR LOAD
AND       K00206	// W10 RH 작업완료 없음
AND NOT   K00210	// W10 RH 파트 로딩완료
OUT       M00214	// W10 RH 파트이상
; L56
LOAD      M00203	// W10 RH 자동기동
AND       M00240	// W10 RH 로보트 간섭무
AND       M00232	// W10 RH 기동 Pulse
AND       M00221	// W10 RH 파트 OK
AND       K00206	// W10 RH 작업완료 없음
AND=      0 D018502	// W10 RH 차종 정보
LOAD      M00215	// W10 RH 차종선택 이상
AND NOT   M00205	// W10 RH 이상해제
OR LOAD
AND       F0009A
OUT       M00215	// W10 RH 차종선택 이상
; L58
LOAD      F0009A
LOAD      M00216	// W10 RH 이상
AND NOT   M00205	// W10 RH 이상해제
OR LOAD
OUT       M00216	// W10 RH 이상
; L60
LOAD      F0009A
LOAD      M00217	// W10 RH 서보이상
AND NOT   M00205	// W10 RH 이상해제
OR LOAD
OUT       M00217	// W10 RH 서보이상

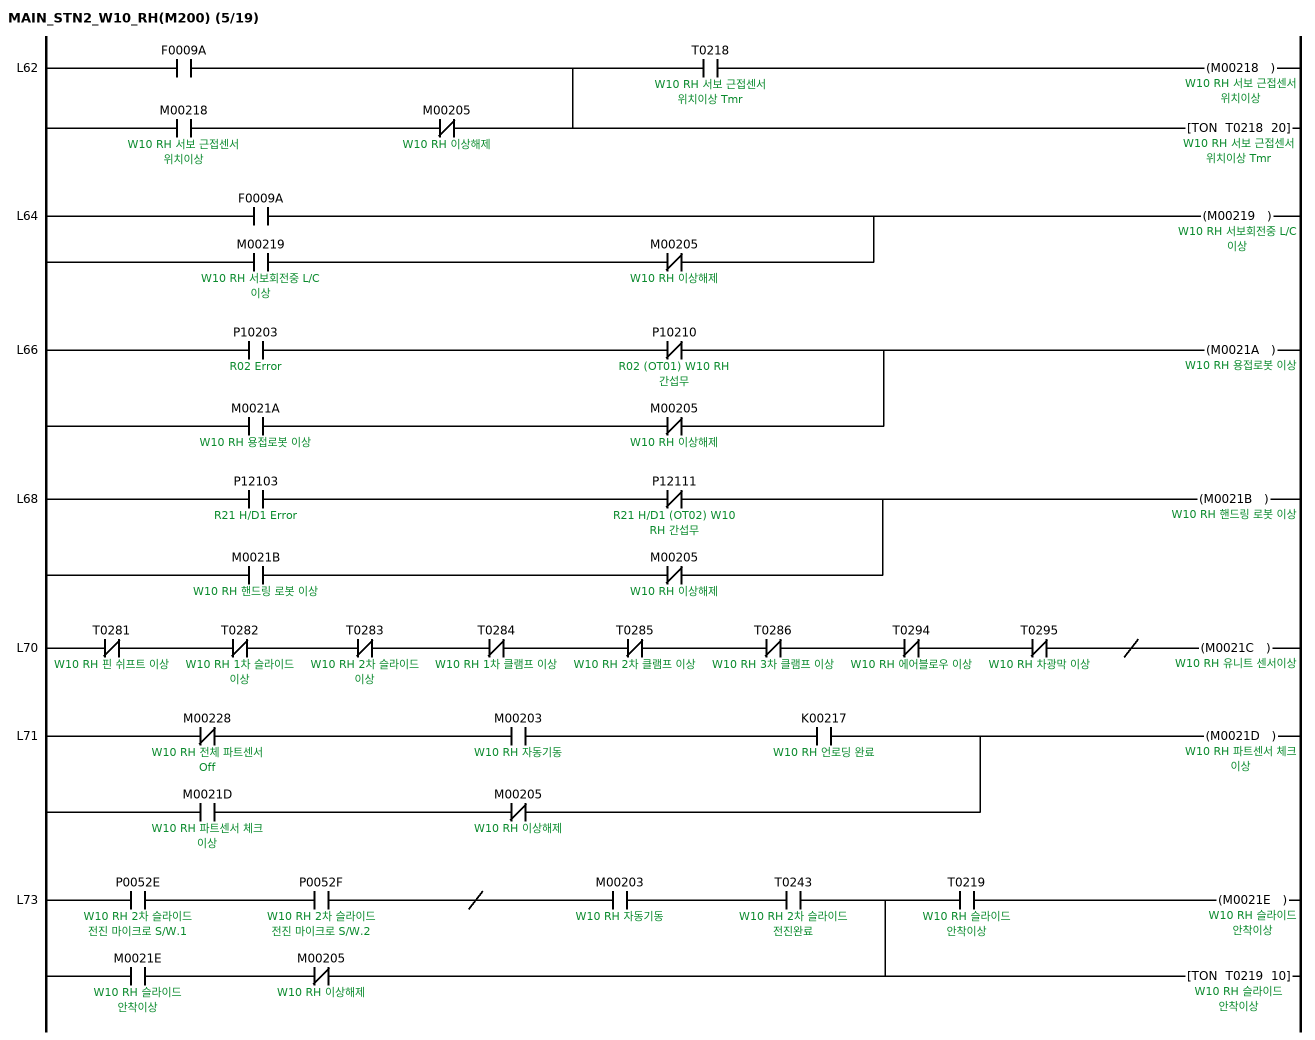
; L62
LOAD      F0009A
LOAD      M00218	// W10 RH 서보 근접센서 위치이상
AND NOT   M00205	// W10 RH 이상해제
OR LOAD
MPUSH
AND       T0218	// W10 RH 서보 근접센서 위치이상 Tmr
OUT       M00218	// W10 RH 서보 근접센서 위치이상
MPOP
TON       T0218 20	// W10 RH 서보 근접센서 위치이상 Tmr
; L64
LOAD      F0009A
LOAD      M00219	// W10 RH 서보회전중 L/C 이상
AND NOT   M00205	// W10 RH 이상해제
OR LOAD
OUT       M00219	// W10 RH 서보회전중 L/C 이상
; L66
LOAD      P10203	// R02 Error
AND NOT   P10210	// R02 (OT01) W10 RH 간섭무
LOAD      M0021A	// W10 RH 용접로봇 이상
AND NOT   M00205	// W10 RH 이상해제
OR LOAD
OUT       M0021A	// W10 RH 용접로봇 이상
; L68
LOAD      P12103	// R21 H/D1 Error
AND NOT   P12111	// R21 H/D1 (OT02) W10 RH 간섭무
LOAD      M0021B	// W10 RH 핸드링 로봇 이상
AND NOT   M00205	// W10 RH 이상해제
OR LOAD
OUT       M0021B	// W10 RH 핸드링 로봇 이상
; L70
LOAD NOT  T0281	// W10 RH 핀 쉬프트 이상
AND NOT   T0282	// W10 RH 1차 슬라이드 이상
AND NOT   T0283	// W10 RH 2차 슬라이드 이상
AND NOT   T0284	// W10 RH 1차 클램프 이상
AND NOT   T0285	// W10 RH 2차 클램프 이상
AND NOT   T0286	// W10 RH 3차 클램프 이상
AND NOT   T0294	// W10 RH 에어블로우 이상
AND NOT   T0295	// W10 RH 차광막 이상
NOT
OUT       M0021C	// W10 RH 유니트 센서이상
; L71
LOAD NOT  M00228	// W10 RH 전체 파트센서 Off
AND       M00203	// W10 RH 자동기동
AND       K00217	// W10 RH 언로딩 완료
LOAD      M0021D	// W10 RH 파트센서 체크 이상
AND NOT   M00205	// W10 RH 이상해제
OR LOAD
OUT       M0021D	// W10 RH 파트센서 체크 이상
; L73
LOAD      P0052E	// W10 RH 2차 슬라이드 전진 마이크로 S/W.1
AND       P0052F	// W10 RH 2차 슬라이드 전진 마이크로 S/W.2
NOT
AND       M00203	// W10 RH 자동기동
AND       T0243	// W10 RH 2차 슬라이드 전진완료
LOAD      M0021E	// W10 RH 슬라이드 안착이상
AND NOT   M00205	// W10 RH 이상해제
OR LOAD
MPUSH
AND       T0219	// W10 RH 슬라이드 안착이상
OUT       M0021E	// W10 RH 슬라이드 안착이상
MPOP
TON       T0219 10	// W10 RH 슬라이드 안착이상

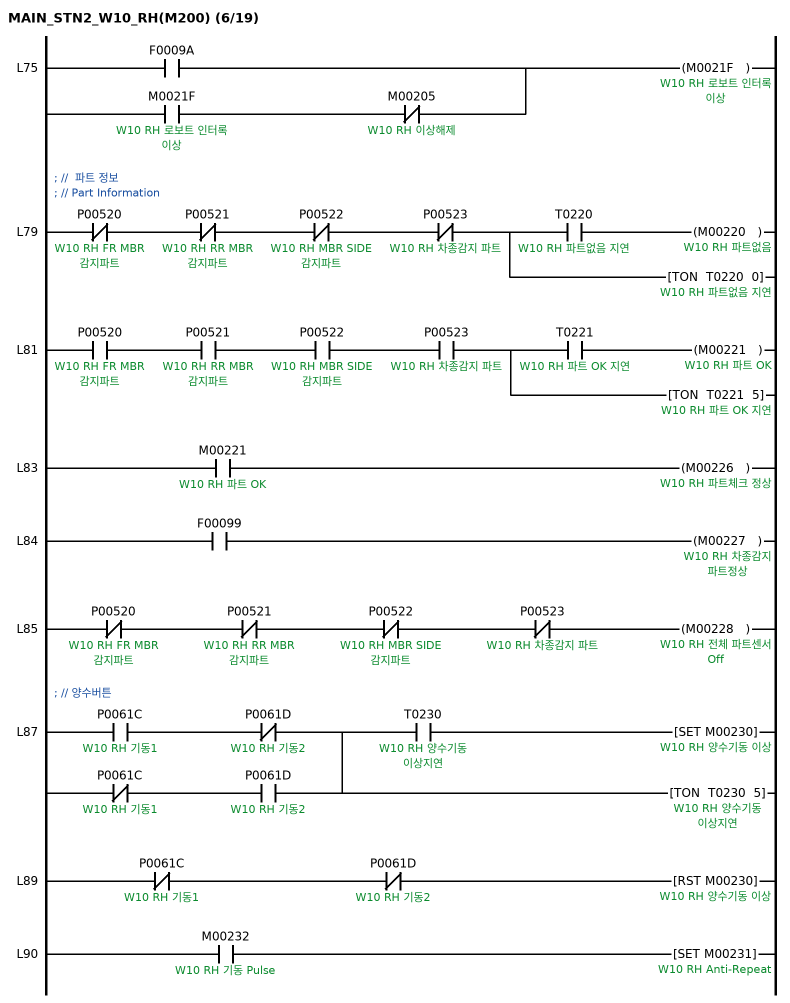
; L75
LOAD      F0009A
LOAD      M0021F	// W10 RH 로보트 인터록 이상
AND NOT   M00205	// W10 RH 이상해제
OR LOAD
OUT       M0021F	// W10 RH 로보트 인터록 이상
//   //  파트 정보
//   // Part Information
; L79
LOAD NOT  P00520	// W10 RH FR MBR 감지파트
AND NOT   P00521	// W10 RH RR MBR 감지파트
AND NOT   P00522	// W10 RH MBR SIDE 감지파트
AND NOT   P00523	// W10 RH 차종감지 파트
MPUSH
AND       T0220	// W10 RH 파트없음 지연
OUT       M00220	// W10 RH 파트없음
MPOP
TON       T0220 0	// W10 RH 파트없음 지연
; L81
LOAD      P00520	// W10 RH FR MBR 감지파트
AND       P00521	// W10 RH RR MBR 감지파트
AND       P00522	// W10 RH MBR SIDE 감지파트
AND       P00523	// W10 RH 차종감지 파트
MPUSH
AND       T0221	// W10 RH 파트 OK 지연
OUT       M00221	// W10 RH 파트 OK
MPOP
TON       T0221 5	// W10 RH 파트 OK 지연
; L83
LOAD      M00221	// W10 RH 파트 OK
OUT       M00226	// W10 RH 파트체크 정상
; L84
LOAD      F00099
OUT       M00227	// W10 RH 차종감지 파트정상
; L85
LOAD NOT  P00520	// W10 RH FR MBR 감지파트
AND NOT   P00521	// W10 RH RR MBR 감지파트
AND NOT   P00522	// W10 RH MBR SIDE 감지파트
AND NOT   P00523	// W10 RH 차종감지 파트
OUT       M00228	// W10 RH 전체 파트센서 Off
//   // 양수버튼
; L87
LOAD      P0061C	// W10 RH 기동1
AND NOT   P0061D	// W10 RH 기동2
LOAD NOT  P0061C	// W10 RH 기동1
AND       P0061D	// W10 RH 기동2
OR LOAD
MPUSH
AND       T0230	// W10 RH 양수기동 이상지연
SET       M00230	// W10 RH 양수기동 이상
MPOP
TON       T0230 5	// W10 RH 양수기동 이상지연
; L89
LOAD NOT  P0061C	// W10 RH 기동1
AND NOT   P0061D	// W10 RH 기동2
RST       M00230	// W10 RH 양수기동 이상
; L90
LOAD      M00232	// W10 RH 기동 Pulse
SET       M00231	// W10 RH Anti-Repeat

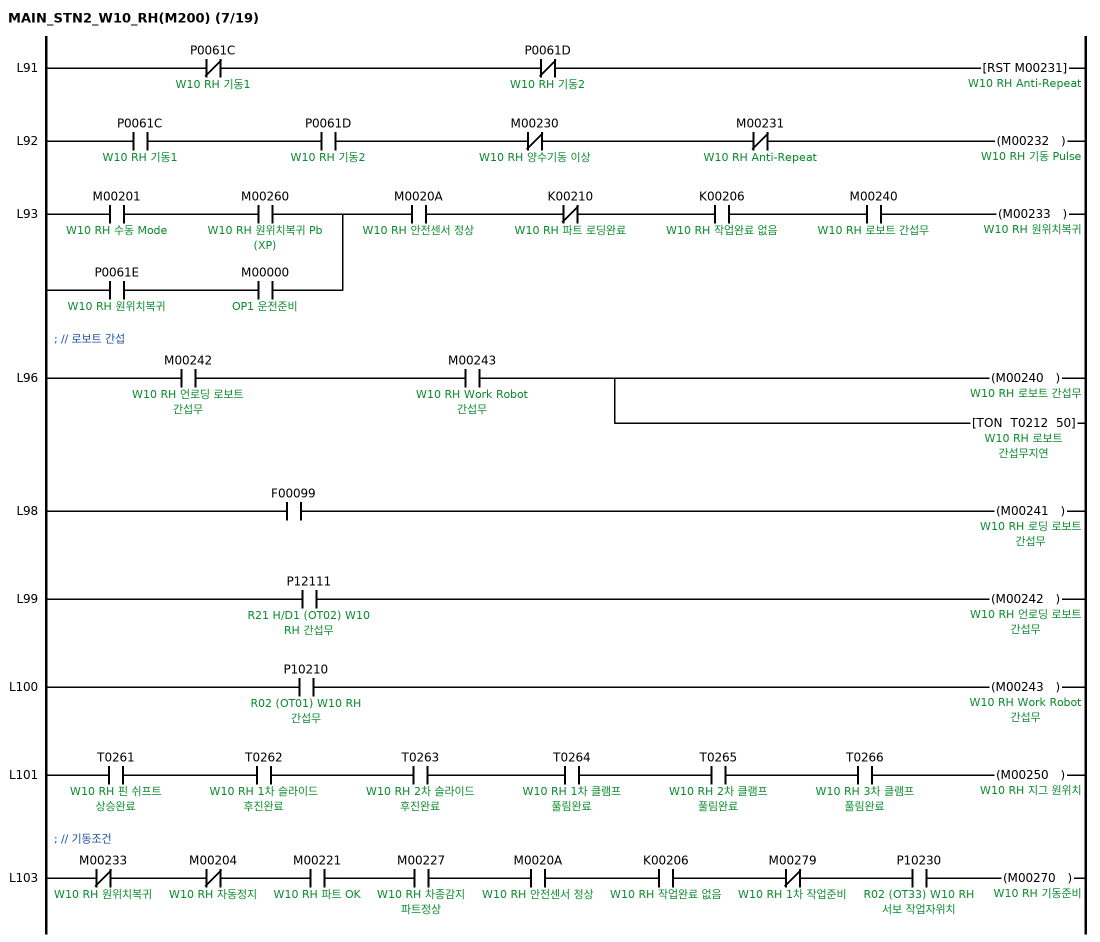
; L91
LOAD NOT  P0061C	// W10 RH 기동1
AND NOT   P0061D	// W10 RH 기동2
RST       M00231	// W10 RH Anti-Repeat
; L92
LOAD      P0061C	// W10 RH 기동1
AND       P0061D	// W10 RH 기동2
AND NOT   M00230	// W10 RH 양수기동 이상
AND NOT   M00231	// W10 RH Anti-Repeat
OUT       M00232	// W10 RH 기동 Pulse
; L93
LOAD      M00201	// W10 RH 수동 Mode
AND       M00260	// W10 RH 원위치복귀 Pb (XP)
LOAD      P0061E	// W10 RH 원위치복귀
AND       M00000	// OP1 운전준비
OR LOAD
AND       M0020A	// W10 RH 안전센서 정상
AND NOT   K00210	// W10 RH 파트 로딩완료
AND       K00206	// W10 RH 작업완료 없음
AND       M00240	// W10 RH 로보트 간섭무
OUT       M00233	// W10 RH 원위치복귀
//   // 로보트 간섭
; L96
LOAD      M00242	// W10 RH 언로딩 로보트 간섭무
AND       M00243	// W10 RH Work Robot 간섭무
OUT       M00240	// W10 RH 로보트 간섭무
TON       T0212 50	// W10 RH 로보트 간섭무지연
; L98
LOAD      F00099
OUT       M00241	// W10 RH 로딩 로보트 간섭무
; L99
LOAD      P12111	// R21 H/D1 (OT02) W10 RH 간섭무
OUT       M00242	// W10 RH 언로딩 로보트 간섭무
; L100
LOAD      P10210	// R02 (OT01) W10 RH 간섭무
OUT       M00243	// W10 RH Work Robot 간섭무
; L101
LOAD      T0261	// W10 RH 핀 쉬프트 상승완료
AND       T0262	// W10 RH 1차 슬라이드 후진완료
AND       T0263	// W10 RH 2차 슬라이드 후진완료
AND       T0264	// W10 RH 1차 클램프 풀림완료
AND       T0265	// W10 RH 2차 클램프 풀림완료
AND       T0266	// W10 RH 3차 클램프 풀림완료
OUT       M00250	// W10 RH 지그 원위치
//   // 기동조건
; L103
LOAD NOT  M00233	// W10 RH 원위치복귀
AND NOT   M00204	// W10 RH 자동정지
AND       M00221	// W10 RH 파트 OK
AND       M00227	// W10 RH 차종감지 파트정상
AND       M0020A	// W10 RH 안전센서 정상
AND       K00206	// W10 RH 작업완료 없음
AND NOT   M00279	// W10 RH 1차 작업준비
AND       P10230	// R02 (OT33) W10 RH 서보 작업자위치
OUT       M00270	// W10 RH 기동준비

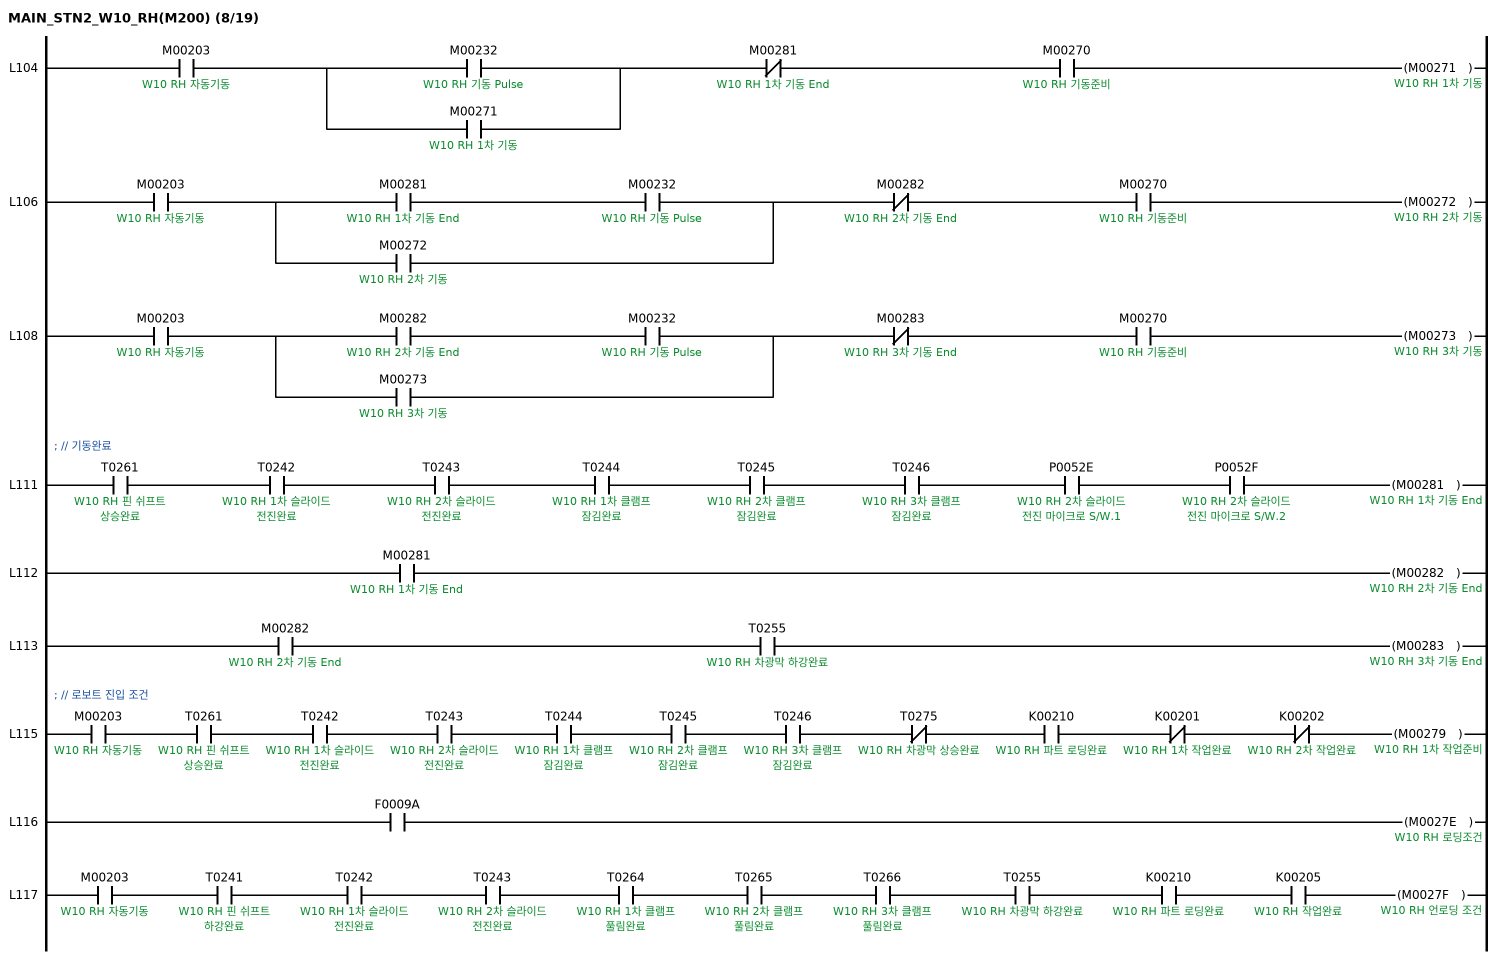
; L104
LOAD      M00203	// W10 RH 자동기동
LOAD      M00232	// W10 RH 기동 Pulse
OR        M00271	// W10 RH 1차 기동
AND LOAD
AND NOT   M00281	// W10 RH 1차 기동 End
AND       M00270	// W10 RH 기동준비
OUT       M00271	// W10 RH 1차 기동
; L106
LOAD      M00203	// W10 RH 자동기동
LOAD      M00281	// W10 RH 1차 기동 End
AND       M00232	// W10 RH 기동 Pulse
OR        M00272	// W10 RH 2차 기동
AND LOAD
AND NOT   M00282	// W10 RH 2차 기동 End
AND       M00270	// W10 RH 기동준비
OUT       M00272	// W10 RH 2차 기동
; L108
LOAD      M00203	// W10 RH 자동기동
LOAD      M00282	// W10 RH 2차 기동 End
AND       M00232	// W10 RH 기동 Pulse
OR        M00273	// W10 RH 3차 기동
AND LOAD
AND NOT   M00283	// W10 RH 3차 기동 End
AND       M00270	// W10 RH 기동준비
OUT       M00273	// W10 RH 3차 기동
//   // 기동완료
; L111
LOAD      T0261	// W10 RH 핀 쉬프트 상승완료
AND       T0242	// W10 RH 1차 슬라이드 전진완료
AND       T0243	// W10 RH 2차 슬라이드 전진완료
AND       T0244	// W10 RH 1차 클램프 잠김완료
AND       T0245	// W10 RH 2차 클램프 잠김완료
AND       T0246	// W10 RH 3차 클램프 잠김완료
AND       P0052E	// W10 RH 2차 슬라이드 전진 마이크로 S/W.1
AND       P0052F	// W10 RH 2차 슬라이드 전진 마이크로 S/W.2
OUT       M00281	// W10 RH 1차 기동 End
; L112
LOAD      M00281	// W10 RH 1차 기동 End
OUT       M00282	// W10 RH 2차 기동 End
; L113
LOAD      M00282	// W10 RH 2차 기동 End
AND       T0255	// W10 RH 차광막 하강완료
OUT       M00283	// W10 RH 3차 기동 End
//   // 로보트 진입 조건
; L115
LOAD      M00203	// W10 RH 자동기동
AND       T0261	// W10 RH 핀 쉬프트 상승완료
AND       T0242	// W10 RH 1차 슬라이드 전진완료
AND       T0243	// W10 RH 2차 슬라이드 전진완료
AND       T0244	// W10 RH 1차 클램프 잠김완료
AND       T0245	// W10 RH 2차 클램프 잠김완료
AND       T0246	// W10 RH 3차 클램프 잠김완료
AND NOT   T0275	// W10 RH 차광막 상승완료
AND       K00210	// W10 RH 파트 로딩완료
AND NOT   K00201	// W10 RH 1차 작업완료
AND NOT   K00202	// W10 RH 2차 작업완료
OUT       M00279	// W10 RH 1차 작업준비
; L116
LOAD      F0009A
OUT       M0027E	// W10 RH 로딩조건
; L117
LOAD      M00203	// W10 RH 자동기동
AND       T0241	// W10 RH 핀 쉬프트 하강완료
AND       T0242	// W10 RH 1차 슬라이드 전진완료
AND       T0243	// W10 RH 2차 슬라이드 전진완료
AND       T0264	// W10 RH 1차 클램프 풀림완료
AND       T0265	// W10 RH 2차 클램프 풀림완료
AND       T0266	// W10 RH 3차 클램프 풀림완료
AND       T0255	// W10 RH 차광막 하강완료
AND       K00210	// W10 RH 파트 로딩완료
AND       K00205	// W10 RH 작업완료
OUT       M0027F	// W10 RH 언로딩 조건

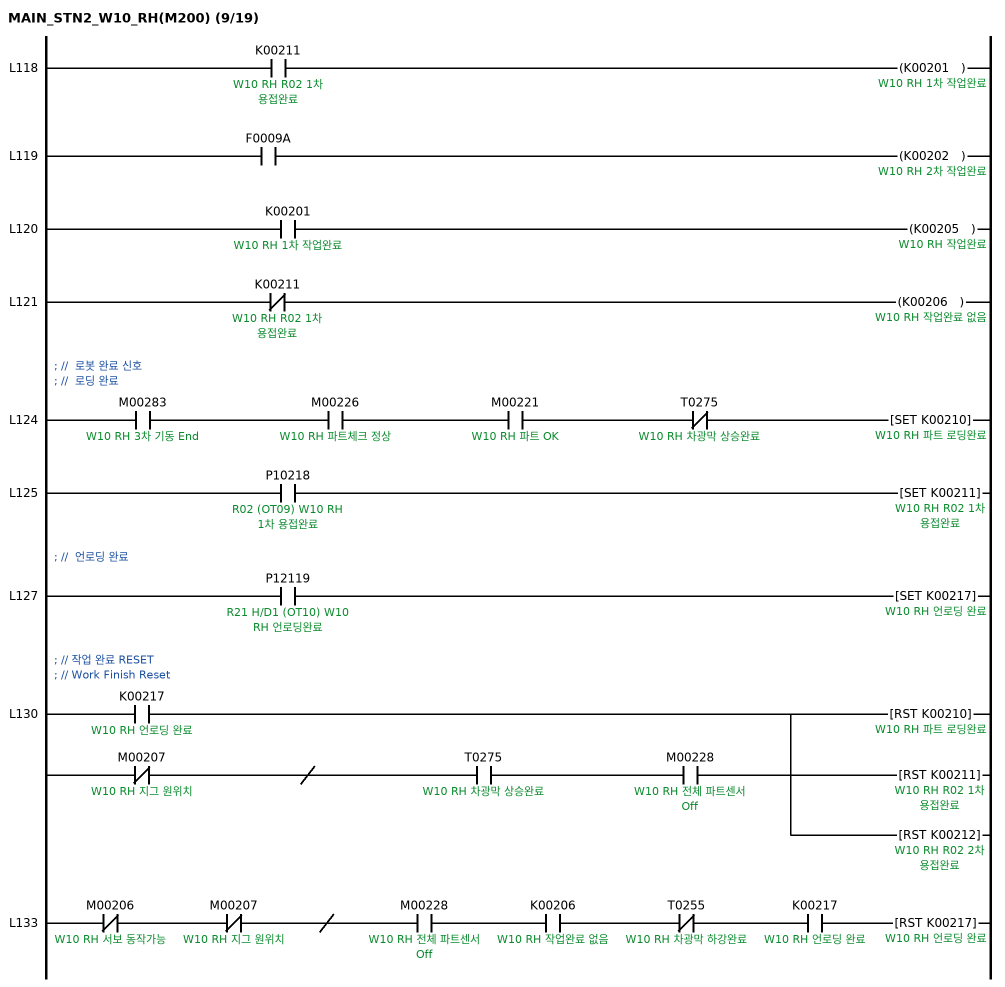
; L118
LOAD      K00211	// W10 RH R02 1차 용접완료
OUT       K00201	// W10 RH 1차 작업완료
; L119
LOAD      F0009A
OUT       K00202	// W10 RH 2차 작업완료
; L120
LOAD      K00201	// W10 RH 1차 작업완료
OUT       K00205	// W10 RH 작업완료
; L121
LOAD NOT  K00211	// W10 RH R02 1차 용접완료
OUT       K00206	// W10 RH 작업완료 없음
//   //  로봇 완료 신호
//   //  로딩 완료
; L124
LOAD      M00283	// W10 RH 3차 기동 End
AND       M00226	// W10 RH 파트체크 정상
AND       M00221	// W10 RH 파트 OK
AND NOT   T0275	// W10 RH 차광막 상승완료
SET       K00210	// W10 RH 파트 로딩완료
; L125
LOAD      P10218	// R02 (OT09) W10 RH 1차 용접완료
SET       K00211	// W10 RH R02 1차 용접완료
//   //  언로딩 완료
; L127
LOAD      P12119	// R21 H/D1 (OT10) W10 RH 언로딩완료
SET       K00217	// W10 RH 언로딩 완료
//     // 작업 완료 RESET
//   // Work Finish Reset
; L130
LOAD      K00217	// W10 RH 언로딩 완료
LOAD NOT  M00207	// W10 RH 지그 원위치
NOT
AND       T0275	// W10 RH 차광막 상승완료
AND       M00228	// W10 RH 전체 파트센서 Off
OR LOAD
RST       K00210	// W10 RH 파트 로딩완료
RST       K00211	// W10 RH R02 1차 용접완료
RST       K00212	// W10 RH R02 2차 용접완료
; L133
LOAD NOT  M00206	// W10 RH 서보 동작가능
AND NOT   M00207	// W10 RH 지그 원위치
NOT
AND       M00228	// W10 RH 전체 파트센서 Off
AND       K00206	// W10 RH 작업완료 없음
AND NOT   T0255	// W10 RH 차광막 하강완료
AND       K00217	// W10 RH 언로딩 완료
RST       K00217	// W10 RH 언로딩 완료

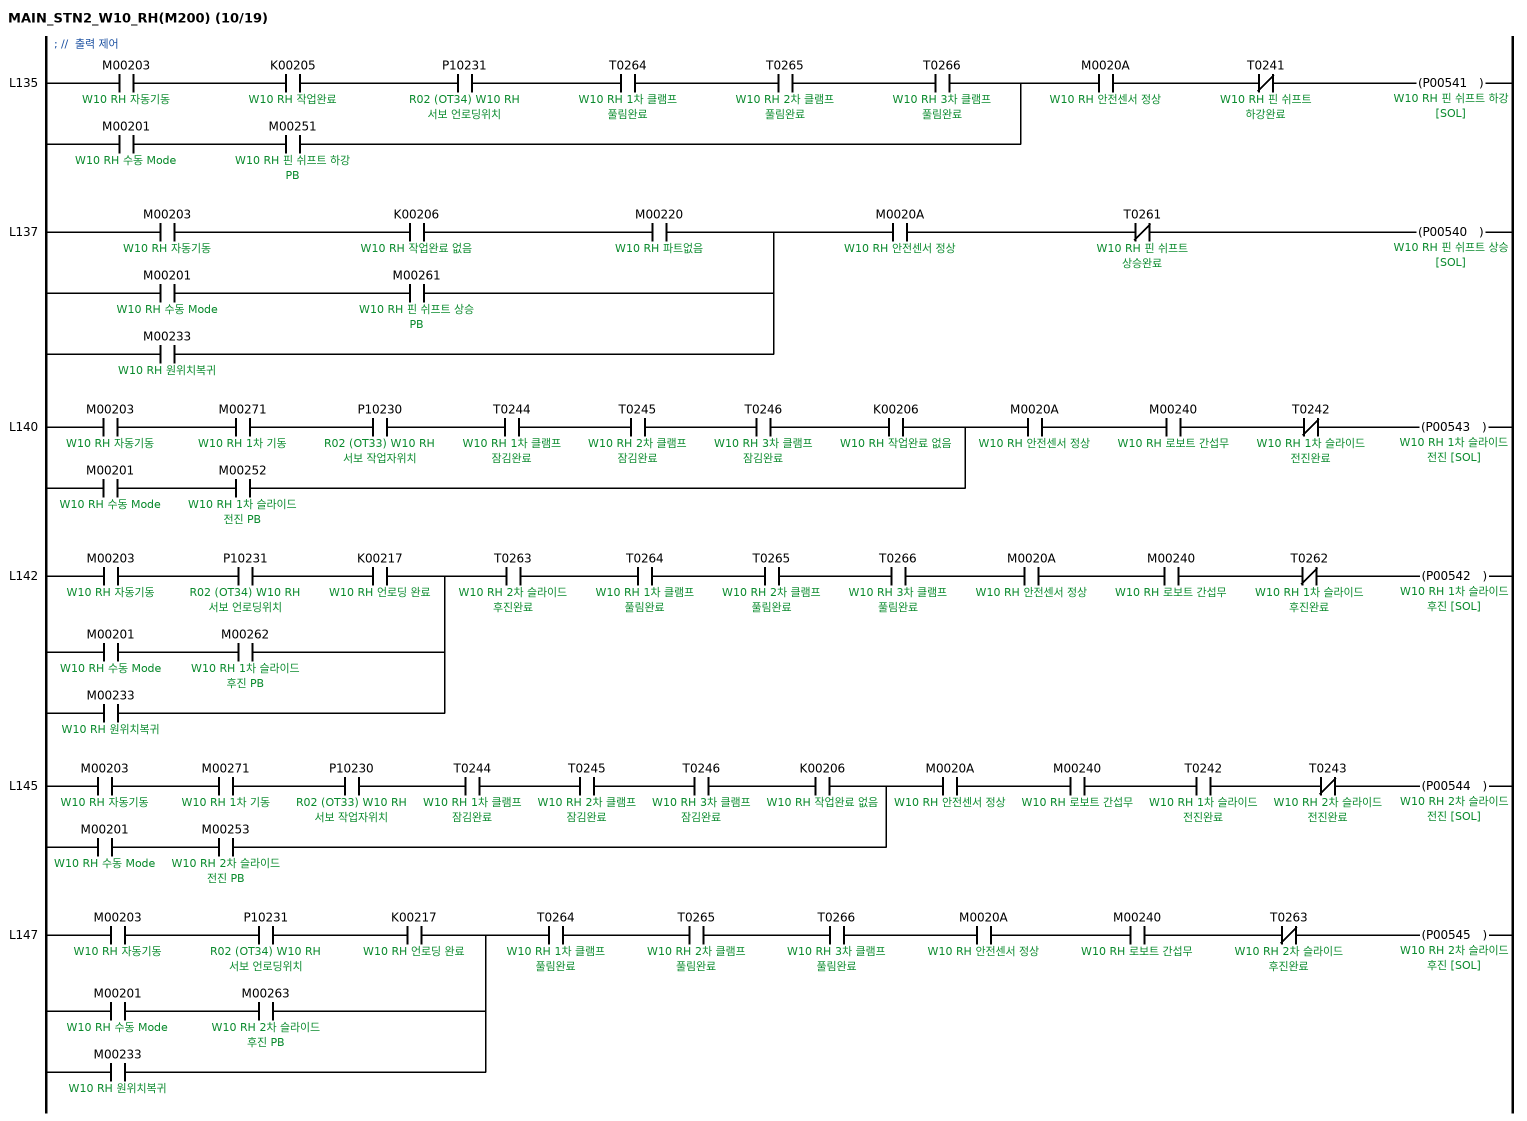
//     //  출력 제어
; L135
LOAD      M00203	// W10 RH 자동기동
AND       K00205	// W10 RH 작업완료
AND       P10231	// R02 (OT34) W10 RH 서보 언로딩위치
AND       T0264	// W10 RH 1차 클램프 풀림완료
AND       T0265	// W10 RH 2차 클램프 풀림완료
AND       T0266	// W10 RH 3차 클램프 풀림완료
LOAD      M00201	// W10 RH 수동 Mode
AND       M00251	// W10 RH 핀 쉬프트 하강 PB
OR LOAD
AND       M0020A	// W10 RH 안전센서 정상
AND NOT   T0241	// W10 RH 핀 쉬프트 하강완료
OUT       P00541	// W10 RH 핀 쉬프트 하강 [SOL]
; L137
LOAD      M00203	// W10 RH 자동기동
AND       K00206	// W10 RH 작업완료 없음
AND       M00220	// W10 RH 파트없음
LOAD      M00201	// W10 RH 수동 Mode
AND       M00261	// W10 RH 핀 쉬프트 상승 PB
OR LOAD
OR        M00233	// W10 RH 원위치복귀
AND       M0020A	// W10 RH 안전센서 정상
AND NOT   T0261	// W10 RH 핀 쉬프트 상승완료
OUT       P00540	// W10 RH 핀 쉬프트 상승 [SOL]
; L140
LOAD      M00203	// W10 RH 자동기동
AND       M00271	// W10 RH 1차 기동
AND       P10230	// R02 (OT33) W10 RH 서보 작업자위치
AND       T0244	// W10 RH 1차 클램프 잠김완료
AND       T0245	// W10 RH 2차 클램프 잠김완료
AND       T0246	// W10 RH 3차 클램프 잠김완료
AND       K00206	// W10 RH 작업완료 없음
LOAD      M00201	// W10 RH 수동 Mode
AND       M00252	// W10 RH 1차 슬라이드 전진 PB
OR LOAD
AND       M0020A	// W10 RH 안전센서 정상
AND       M00240	// W10 RH 로보트 간섭무
AND NOT   T0242	// W10 RH 1차 슬라이드 전진완료
OUT       P00543	// W10 RH 1차 슬라이드 전진 [SOL]
; L142
LOAD      M00203	// W10 RH 자동기동
AND       P10231	// R02 (OT34) W10 RH 서보 언로딩위치
AND       K00217	// W10 RH 언로딩 완료
LOAD      M00201	// W10 RH 수동 Mode
AND       M00262	// W10 RH 1차 슬라이드 후진 PB
OR LOAD
OR        M00233	// W10 RH 원위치복귀
AND       T0263	// W10 RH 2차 슬라이드 후진완료
AND       T0264	// W10 RH 1차 클램프 풀림완료
AND       T0265	// W10 RH 2차 클램프 풀림완료
AND       T0266	// W10 RH 3차 클램프 풀림완료
AND       M0020A	// W10 RH 안전센서 정상
AND       M00240	// W10 RH 로보트 간섭무
AND NOT   T0262	// W10 RH 1차 슬라이드 후진완료
OUT       P00542	// W10 RH 1차 슬라이드 후진 [SOL]
; L145
LOAD      M00203	// W10 RH 자동기동
AND       M00271	// W10 RH 1차 기동
AND       P10230	// R02 (OT33) W10 RH 서보 작업자위치
AND       T0244	// W10 RH 1차 클램프 잠김완료
AND       T0245	// W10 RH 2차 클램프 잠김완료
AND       T0246	// W10 RH 3차 클램프 잠김완료
AND       K00206	// W10 RH 작업완료 없음
LOAD      M00201	// W10 RH 수동 Mode
AND       M00253	// W10 RH 2차 슬라이드 전진 PB
OR LOAD
AND       M0020A	// W10 RH 안전센서 정상
AND       M00240	// W10 RH 로보트 간섭무
AND       T0242	// W10 RH 1차 슬라이드 전진완료
AND NOT   T0243	// W10 RH 2차 슬라이드 전진완료
OUT       P00544	// W10 RH 2차 슬라이드 전진 [SOL]
; L147
LOAD      M00203	// W10 RH 자동기동
AND       P10231	// R02 (OT34) W10 RH 서보 언로딩위치
AND       K00217	// W10 RH 언로딩 완료
LOAD      M00201	// W10 RH 수동 Mode
AND       M00263	// W10 RH 2차 슬라이드 후진 PB
OR LOAD
OR        M00233	// W10 RH 원위치복귀
AND       T0264	// W10 RH 1차 클램프 풀림완료
AND       T0265	// W10 RH 2차 클램프 풀림완료
AND       T0266	// W10 RH 3차 클램프 풀림완료
AND       M0020A	// W10 RH 안전센서 정상
AND       M00240	// W10 RH 로보트 간섭무
AND NOT   T0263	// W10 RH 2차 슬라이드 후진완료
OUT       P00545	// W10 RH 2차 슬라이드 후진 [SOL]

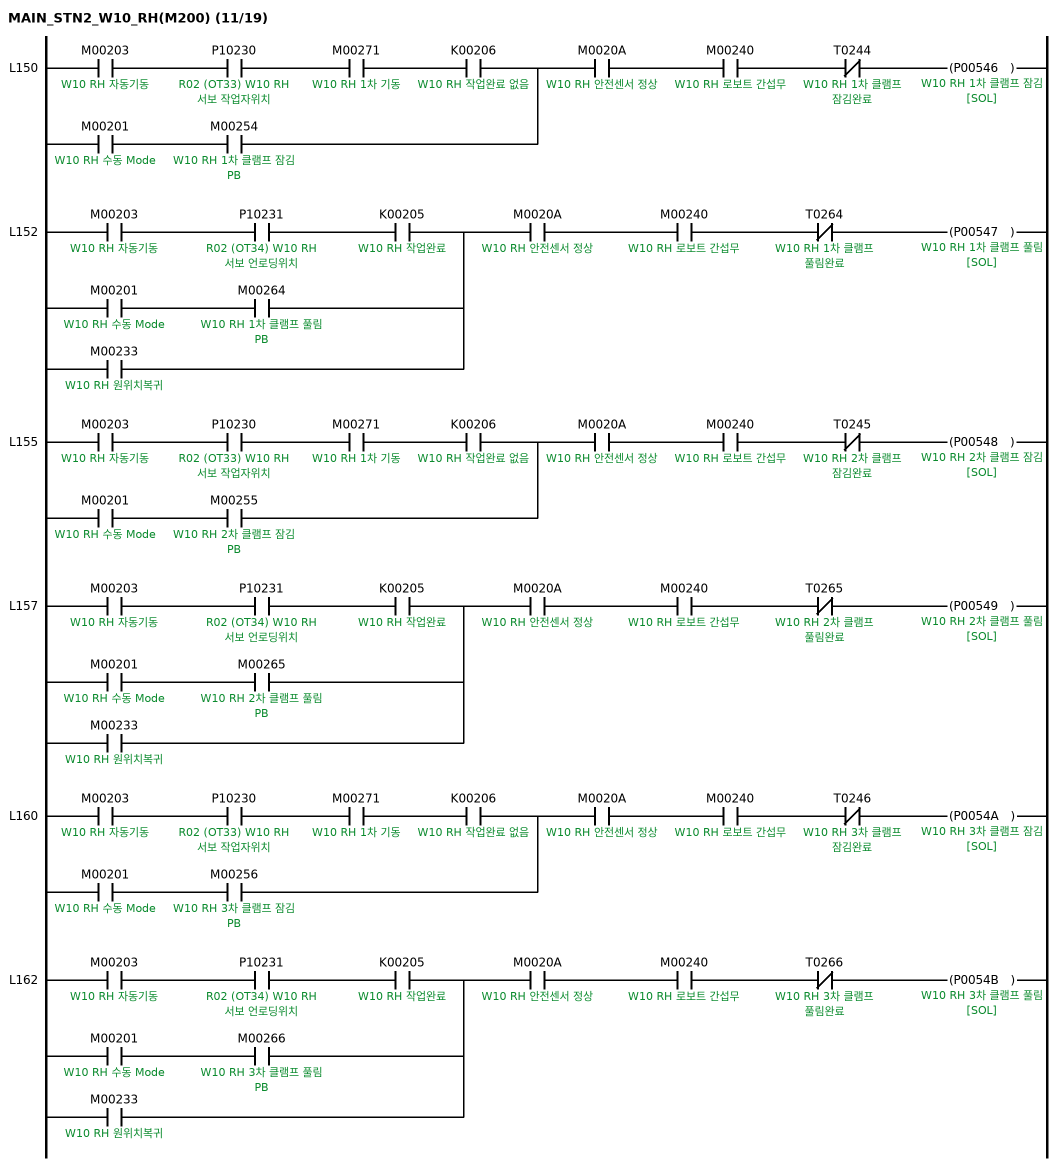
; L150
LOAD      M00203	// W10 RH 자동기동
AND       P10230	// R02 (OT33) W10 RH 서보 작업자위치
AND       M00271	// W10 RH 1차 기동
AND       K00206	// W10 RH 작업완료 없음
LOAD      M00201	// W10 RH 수동 Mode
AND       M00254	// W10 RH 1차 클램프 잠김 PB
OR LOAD
AND       M0020A	// W10 RH 안전센서 정상
AND       M00240	// W10 RH 로보트 간섭무
AND NOT   T0244	// W10 RH 1차 클램프 잠김완료
OUT       P00546	// W10 RH 1차 클램프 잠김 [SOL]
; L152
LOAD      M00203	// W10 RH 자동기동
AND       P10231	// R02 (OT34) W10 RH 서보 언로딩위치
AND       K00205	// W10 RH 작업완료
LOAD      M00201	// W10 RH 수동 Mode
AND       M00264	// W10 RH 1차 클램프 풀림 PB
OR LOAD
OR        M00233	// W10 RH 원위치복귀
AND       M0020A	// W10 RH 안전센서 정상
AND       M00240	// W10 RH 로보트 간섭무
AND NOT   T0264	// W10 RH 1차 클램프 풀림완료
OUT       P00547	// W10 RH 1차 클램프 풀림 [SOL]
; L155
LOAD      M00203	// W10 RH 자동기동
AND       P10230	// R02 (OT33) W10 RH 서보 작업자위치
AND       M00271	// W10 RH 1차 기동
AND       K00206	// W10 RH 작업완료 없음
LOAD      M00201	// W10 RH 수동 Mode
AND       M00255	// W10 RH 2차 클램프 잠김 PB
OR LOAD
AND       M0020A	// W10 RH 안전센서 정상
AND       M00240	// W10 RH 로보트 간섭무
AND NOT   T0245	// W10 RH 2차 클램프 잠김완료
OUT       P00548	// W10 RH 2차 클램프 잠김 [SOL]
; L157
LOAD      M00203	// W10 RH 자동기동
AND       P10231	// R02 (OT34) W10 RH 서보 언로딩위치
AND       K00205	// W10 RH 작업완료
LOAD      M00201	// W10 RH 수동 Mode
AND       M00265	// W10 RH 2차 클램프 풀림 PB
OR LOAD
OR        M00233	// W10 RH 원위치복귀
AND       M0020A	// W10 RH 안전센서 정상
AND       M00240	// W10 RH 로보트 간섭무
AND NOT   T0265	// W10 RH 2차 클램프 풀림완료
OUT       P00549	// W10 RH 2차 클램프 풀림 [SOL]
; L160
LOAD      M00203	// W10 RH 자동기동
AND       P10230	// R02 (OT33) W10 RH 서보 작업자위치
AND       M00271	// W10 RH 1차 기동
AND       K00206	// W10 RH 작업완료 없음
LOAD      M00201	// W10 RH 수동 Mode
AND       M00256	// W10 RH 3차 클램프 잠김 PB
OR LOAD
AND       M0020A	// W10 RH 안전센서 정상
AND       M00240	// W10 RH 로보트 간섭무
AND NOT   T0246	// W10 RH 3차 클램프 잠김완료
OUT       P0054A	// W10 RH 3차 클램프 잠김 [SOL]
; L162
LOAD      M00203	// W10 RH 자동기동
AND       P10231	// R02 (OT34) W10 RH 서보 언로딩위치
AND       K00205	// W10 RH 작업완료
LOAD      M00201	// W10 RH 수동 Mode
AND       M00266	// W10 RH 3차 클램프 풀림 PB
OR LOAD
OR        M00233	// W10 RH 원위치복귀
AND       M0020A	// W10 RH 안전센서 정상
AND       M00240	// W10 RH 로보트 간섭무
AND NOT   T0266	// W10 RH 3차 클램프 풀림완료
OUT       P0054B	// W10 RH 3차 클램프 풀림 [SOL]

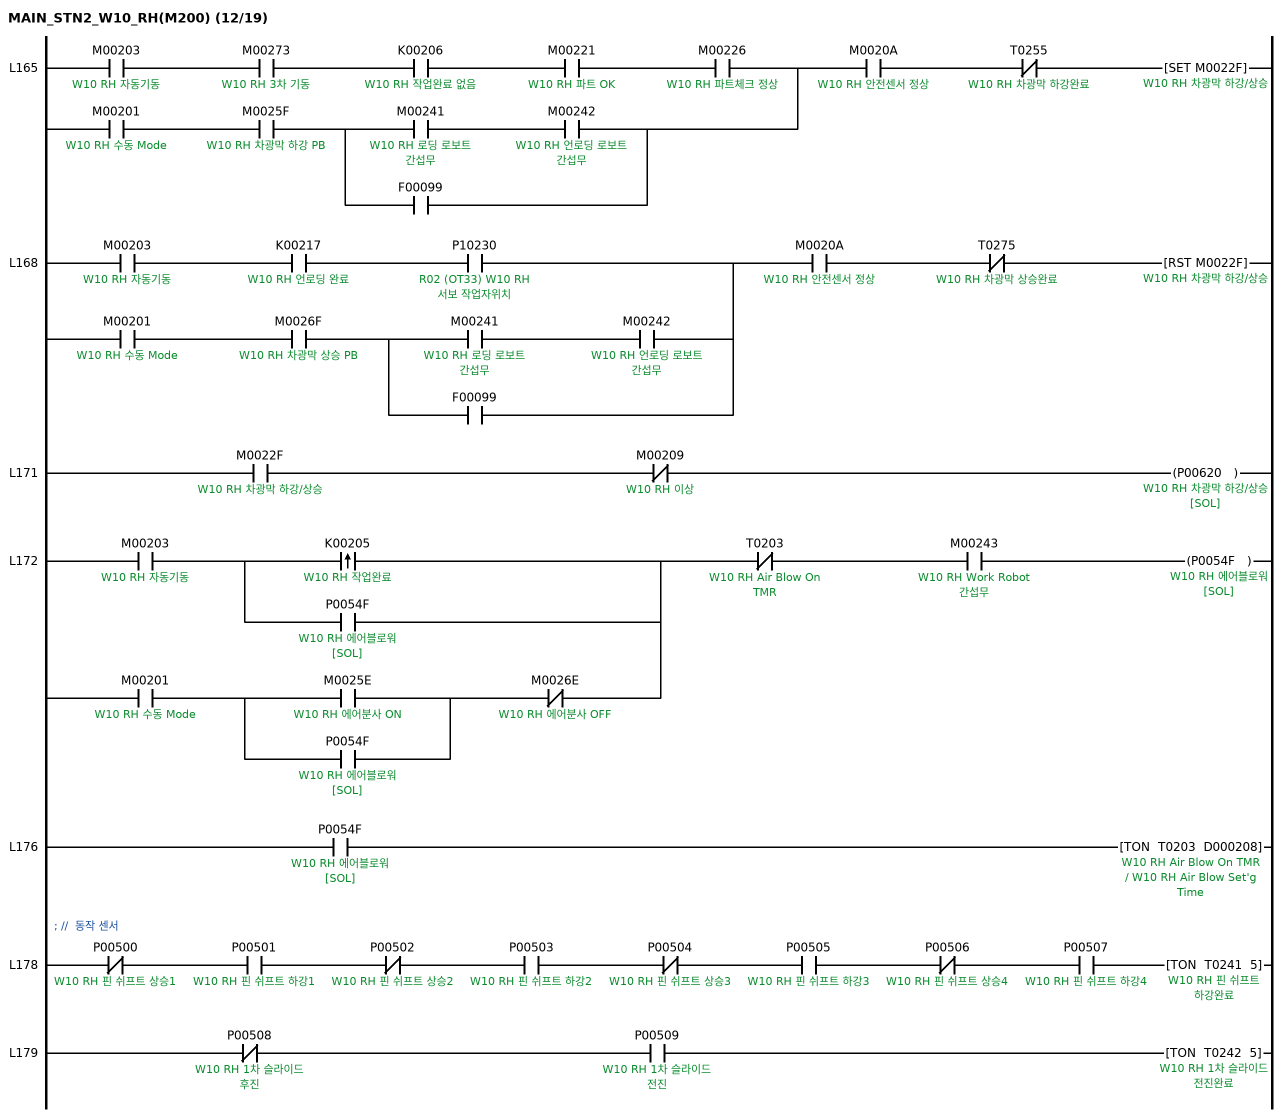
; L165
LOAD      M00203	// W10 RH 자동기동
AND       M00273	// W10 RH 3차 기동
AND       K00206	// W10 RH 작업완료 없음
AND       M00221	// W10 RH 파트 OK
AND       M00226	// W10 RH 파트체크 정상
LOAD      M00201	// W10 RH 수동 Mode
AND       M0025F	// W10 RH 차광막 하강 PB
LOAD      M00241	// W10 RH 로딩 로보트 간섭무
AND       M00242	// W10 RH 언로딩 로보트 간섭무
OR        F00099
AND LOAD
OR LOAD
AND       M0020A	// W10 RH 안전센서 정상
AND NOT   T0255	// W10 RH 차광막 하강완료
SET       M0022F	// W10 RH 차광막 하강/상승
; L168
LOAD      M00203	// W10 RH 자동기동
AND       K00217	// W10 RH 언로딩 완료
AND       P10230	// R02 (OT33) W10 RH 서보 작업자위치
LOAD      M00201	// W10 RH 수동 Mode
AND       M0026F	// W10 RH 차광막 상승 PB
LOAD      M00241	// W10 RH 로딩 로보트 간섭무
AND       M00242	// W10 RH 언로딩 로보트 간섭무
OR        F00099
AND LOAD
OR LOAD
AND       M0020A	// W10 RH 안전센서 정상
AND NOT   T0275	// W10 RH 차광막 상승완료
RST       M0022F	// W10 RH 차광막 하강/상승
; L171
LOAD      M0022F	// W10 RH 차광막 하강/상승
AND NOT   M00209	// W10 RH 이상
OUT       P00620	// W10 RH 차광막 하강/상승 [SOL]
; L172
LOAD      M00203	// W10 RH 자동기동
LOADP     K00205	// W10 RH 작업완료
OR        P0054F	// W10 RH 에어블로워 [SOL]
AND LOAD
LOAD      M00201	// W10 RH 수동 Mode
LOAD      M0025E	// W10 RH 에어분사 ON
OR        P0054F	// W10 RH 에어블로워 [SOL]
AND LOAD
AND NOT   M0026E	// W10 RH 에어분사 OFF
OR LOAD
AND NOT   T0203	// W10 RH Air Blow On TMR
AND       M00243	// W10 RH Work Robot 간섭무
OUT       P0054F	// W10 RH 에어블로워 [SOL]
; L176
LOAD      P0054F	// W10 RH 에어블로워 [SOL]
TON       T0203 D000208	// W10 RH Air Blow On TMR / W10 RH Air Blow Set'g Time
//   //  동작 센서
; L178
LOAD NOT  P00500	// W10 RH 핀 쉬프트 상승1
AND       P00501	// W10 RH 핀 쉬프트 하강1
AND NOT   P00502	// W10 RH 핀 쉬프트 상승2
AND       P00503	// W10 RH 핀 쉬프트 하강2
AND NOT   P00504	// W10 RH 핀 쉬프트 상승3
AND       P00505	// W10 RH 핀 쉬프트 하강3
AND NOT   P00506	// W10 RH 핀 쉬프트 상승4
AND       P00507	// W10 RH 핀 쉬프트 하강4
TON       T0241 5	// W10 RH 핀 쉬프트 하강완료
; L179
LOAD NOT  P00508	// W10 RH 1차 슬라이드 후진
AND       P00509	// W10 RH 1차 슬라이드 전진
TON       T0242 5	// W10 RH 1차 슬라이드 전진완료

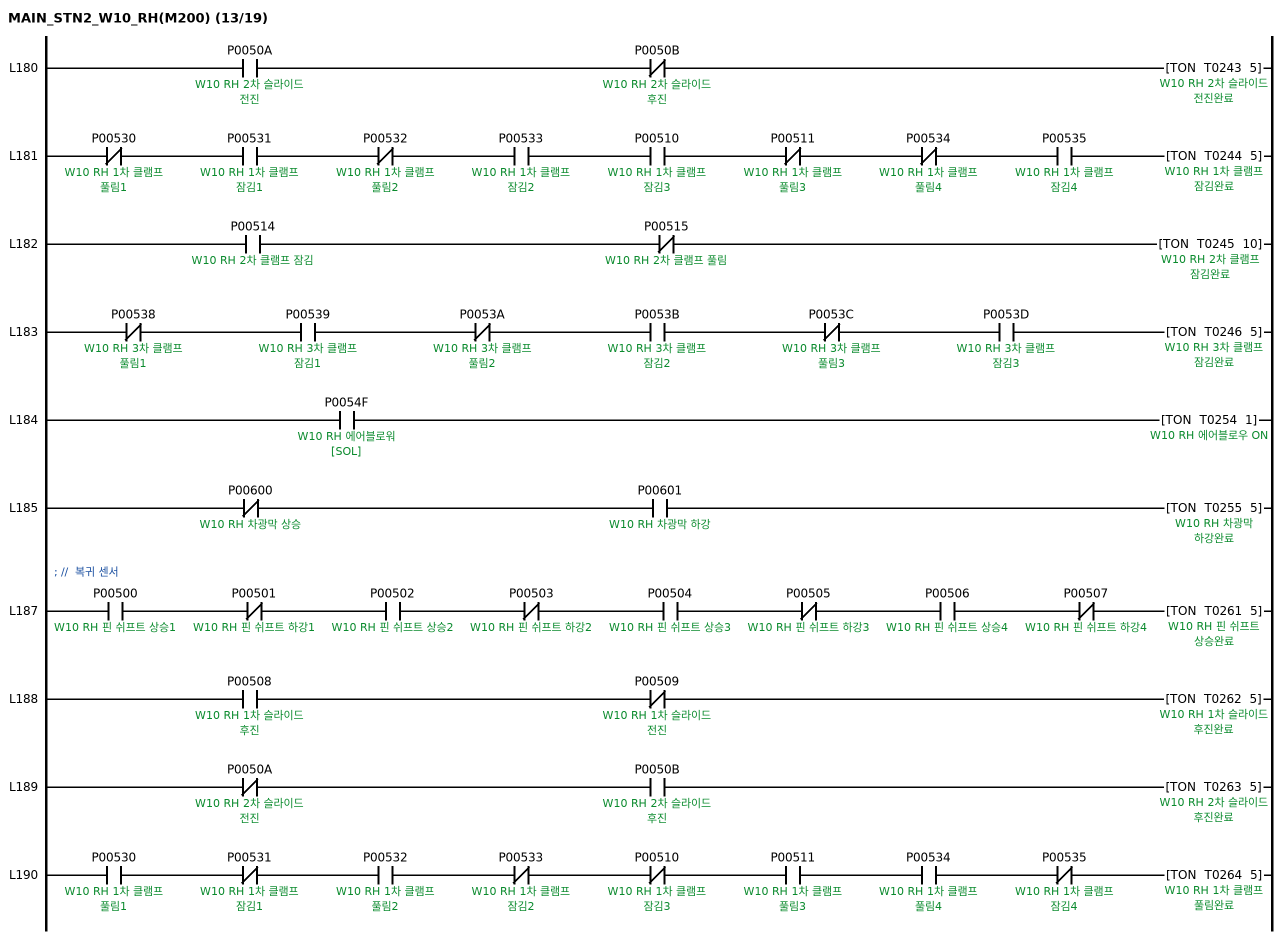
; L180
LOAD      P0050A	// W10 RH 2차 슬라이드 전진
AND NOT   P0050B	// W10 RH 2차 슬라이드 후진
TON       T0243 5	// W10 RH 2차 슬라이드 전진완료
; L181
LOAD NOT  P00530	// W10 RH 1차 클램프 풀림1
AND       P00531	// W10 RH 1차 클램프 잠김1
AND NOT   P00532	// W10 RH 1차 클램프 풀림2
AND       P00533	// W10 RH 1차 클램프 잠김2
AND       P00510	// W10 RH 1차 클램프 잠김3
AND NOT   P00511	// W10 RH 1차 클램프 풀림3
AND NOT   P00534	// W10 RH 1차 클램프 풀림4
AND       P00535	// W10 RH 1차 클램프 잠김4
TON       T0244 5	// W10 RH 1차 클램프 잠김완료
; L182
LOAD      P00514	// W10 RH 2차 클램프 잠김
AND NOT   P00515	// W10 RH 2차 클램프 풀림
TON       T0245 10	// W10 RH 2차 클램프 잠김완료
; L183
LOAD NOT  P00538	// W10 RH 3차 클램프 풀림1
AND       P00539	// W10 RH 3차 클램프 잠김1
AND NOT   P0053A	// W10 RH 3차 클램프 풀림2
AND       P0053B	// W10 RH 3차 클램프 잠김2
AND NOT   P0053C	// W10 RH 3차 클램프 풀림3
AND       P0053D	// W10 RH 3차 클램프 잠김3
TON       T0246 5	// W10 RH 3차 클램프 잠김완료
; L184
LOAD      P0054F	// W10 RH 에어블로워 [SOL]
TON       T0254 1	// W10 RH 에어블로우 ON
; L185
LOAD NOT  P00600	// W10 RH 차광막 상승
AND       P00601	// W10 RH 차광막 하강
TON       T0255 5	// W10 RH 차광막 하강완료
//   //  복귀 센서
; L187
LOAD      P00500	// W10 RH 핀 쉬프트 상승1
AND NOT   P00501	// W10 RH 핀 쉬프트 하강1
AND       P00502	// W10 RH 핀 쉬프트 상승2
AND NOT   P00503	// W10 RH 핀 쉬프트 하강2
AND       P00504	// W10 RH 핀 쉬프트 상승3
AND NOT   P00505	// W10 RH 핀 쉬프트 하강3
AND       P00506	// W10 RH 핀 쉬프트 상승4
AND NOT   P00507	// W10 RH 핀 쉬프트 하강4
TON       T0261 5	// W10 RH 핀 쉬프트 상승완료
; L188
LOAD      P00508	// W10 RH 1차 슬라이드 후진
AND NOT   P00509	// W10 RH 1차 슬라이드 전진
TON       T0262 5	// W10 RH 1차 슬라이드 후진완료
; L189
LOAD NOT  P0050A	// W10 RH 2차 슬라이드 전진
AND       P0050B	// W10 RH 2차 슬라이드 후진
TON       T0263 5	// W10 RH 2차 슬라이드 후진완료
; L190
LOAD      P00530	// W10 RH 1차 클램프 풀림1
AND NOT   P00531	// W10 RH 1차 클램프 잠김1
AND       P00532	// W10 RH 1차 클램프 풀림2
AND NOT   P00533	// W10 RH 1차 클램프 잠김2
AND NOT   P00510	// W10 RH 1차 클램프 잠김3
AND       P00511	// W10 RH 1차 클램프 풀림3
AND       P00534	// W10 RH 1차 클램프 풀림4
AND NOT   P00535	// W10 RH 1차 클램프 잠김4
TON       T0264 5	// W10 RH 1차 클램프 풀림완료

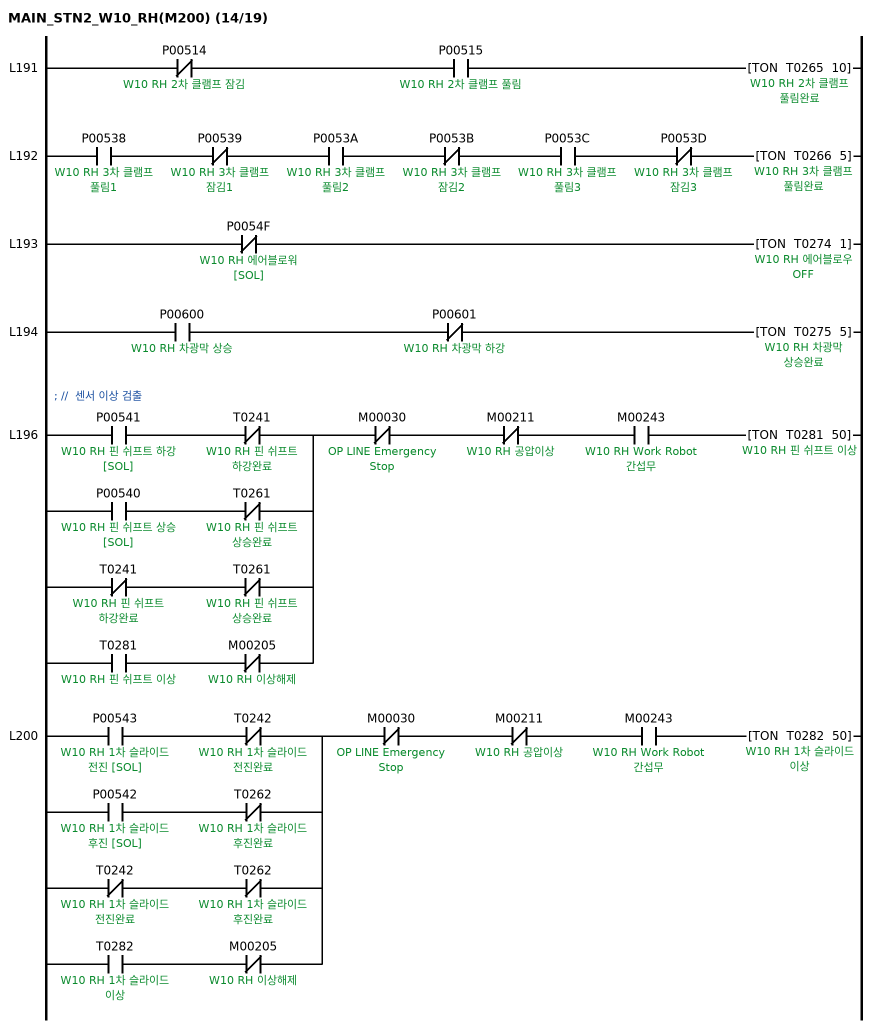
; L191
LOAD NOT  P00514	// W10 RH 2차 클램프 잠김
AND       P00515	// W10 RH 2차 클램프 풀림
TON       T0265 10	// W10 RH 2차 클램프 풀림완료
; L192
LOAD      P00538	// W10 RH 3차 클램프 풀림1
AND NOT   P00539	// W10 RH 3차 클램프 잠김1
AND       P0053A	// W10 RH 3차 클램프 풀림2
AND NOT   P0053B	// W10 RH 3차 클램프 잠김2
AND       P0053C	// W10 RH 3차 클램프 풀림3
AND NOT   P0053D	// W10 RH 3차 클램프 잠김3
TON       T0266 5	// W10 RH 3차 클램프 풀림완료
; L193
LOAD NOT  P0054F	// W10 RH 에어블로워 [SOL]
TON       T0274 1	// W10 RH 에어블로우 OFF
; L194
LOAD      P00600	// W10 RH 차광막 상승
AND NOT   P00601	// W10 RH 차광막 하강
TON       T0275 5	// W10 RH 차광막 상승완료
//     //  센서 이상 검출
; L196
LOAD      P00541	// W10 RH 핀 쉬프트 하강 [SOL]
AND NOT   T0241	// W10 RH 핀 쉬프트 하강완료
LOAD      P00540	// W10 RH 핀 쉬프트 상승 [SOL]
AND NOT   T0261	// W10 RH 핀 쉬프트 상승완료
OR LOAD
LOAD NOT  T0241	// W10 RH 핀 쉬프트 하강완료
AND NOT   T0261	// W10 RH 핀 쉬프트 상승완료
OR LOAD
LOAD      T0281	// W10 RH 핀 쉬프트 이상
AND NOT   M00205	// W10 RH 이상해제
OR LOAD
AND NOT   M00030	// OP LINE Emergency Stop
AND NOT   M00211	// W10 RH 공압이상
AND       M00243	// W10 RH Work Robot 간섭무
TON       T0281 50	// W10 RH 핀 쉬프트 이상
; L200
LOAD      P00543	// W10 RH 1차 슬라이드 전진 [SOL]
AND NOT   T0242	// W10 RH 1차 슬라이드 전진완료
LOAD      P00542	// W10 RH 1차 슬라이드 후진 [SOL]
AND NOT   T0262	// W10 RH 1차 슬라이드 후진완료
OR LOAD
LOAD NOT  T0242	// W10 RH 1차 슬라이드 전진완료
AND NOT   T0262	// W10 RH 1차 슬라이드 후진완료
OR LOAD
LOAD      T0282	// W10 RH 1차 슬라이드 이상
AND NOT   M00205	// W10 RH 이상해제
OR LOAD
AND NOT   M00030	// OP LINE Emergency Stop
AND NOT   M00211	// W10 RH 공압이상
AND       M00243	// W10 RH Work Robot 간섭무
TON       T0282 50	// W10 RH 1차 슬라이드 이상

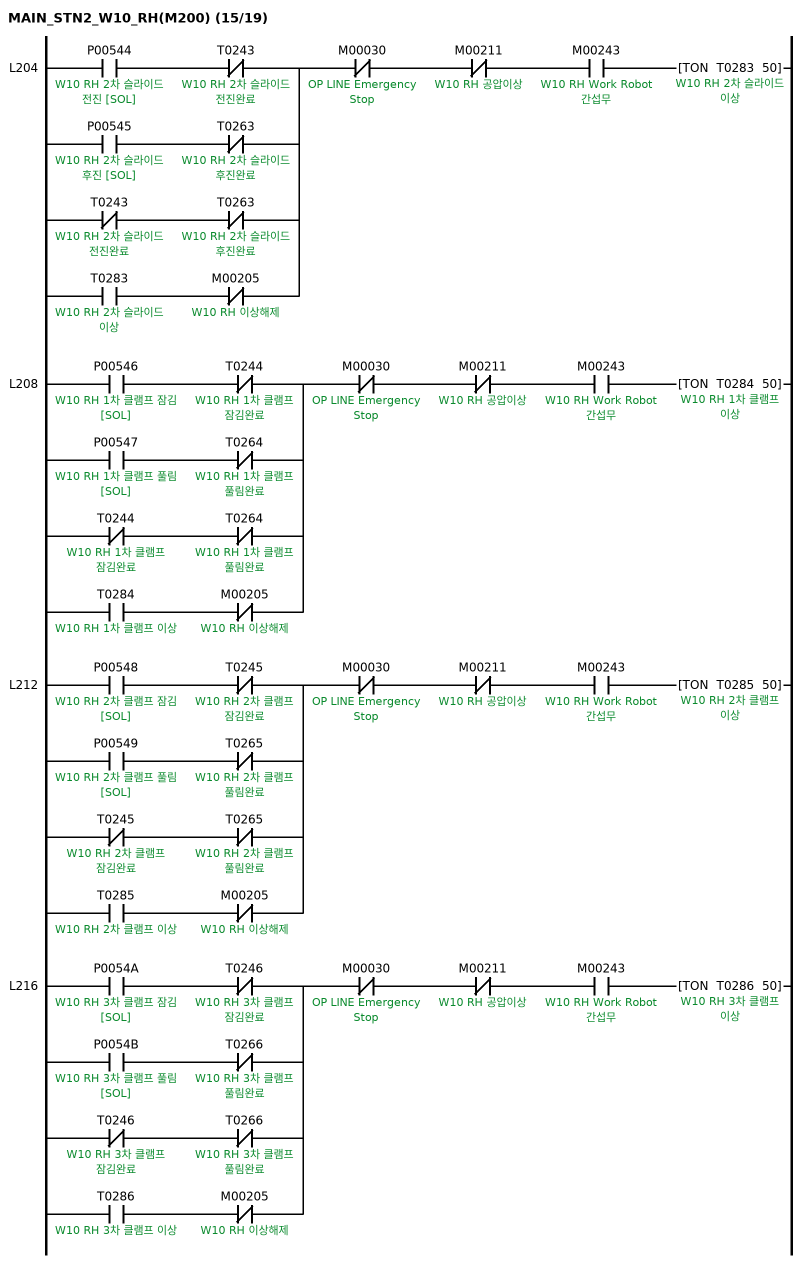
; L204
LOAD      P00544	// W10 RH 2차 슬라이드 전진 [SOL]
AND NOT   T0243	// W10 RH 2차 슬라이드 전진완료
LOAD      P00545	// W10 RH 2차 슬라이드 후진 [SOL]
AND NOT   T0263	// W10 RH 2차 슬라이드 후진완료
OR LOAD
LOAD NOT  T0243	// W10 RH 2차 슬라이드 전진완료
AND NOT   T0263	// W10 RH 2차 슬라이드 후진완료
OR LOAD
LOAD      T0283	// W10 RH 2차 슬라이드 이상
AND NOT   M00205	// W10 RH 이상해제
OR LOAD
AND NOT   M00030	// OP LINE Emergency Stop
AND NOT   M00211	// W10 RH 공압이상
AND       M00243	// W10 RH Work Robot 간섭무
TON       T0283 50	// W10 RH 2차 슬라이드 이상
; L208
LOAD      P00546	// W10 RH 1차 클램프 잠김 [SOL]
AND NOT   T0244	// W10 RH 1차 클램프 잠김완료
LOAD      P00547	// W10 RH 1차 클램프 풀림 [SOL]
AND NOT   T0264	// W10 RH 1차 클램프 풀림완료
OR LOAD
LOAD NOT  T0244	// W10 RH 1차 클램프 잠김완료
AND NOT   T0264	// W10 RH 1차 클램프 풀림완료
OR LOAD
LOAD      T0284	// W10 RH 1차 클램프 이상
AND NOT   M00205	// W10 RH 이상해제
OR LOAD
AND NOT   M00030	// OP LINE Emergency Stop
AND NOT   M00211	// W10 RH 공압이상
AND       M00243	// W10 RH Work Robot 간섭무
TON       T0284 50	// W10 RH 1차 클램프 이상
; L212
LOAD      P00548	// W10 RH 2차 클램프 잠김 [SOL]
AND NOT   T0245	// W10 RH 2차 클램프 잠김완료
LOAD      P00549	// W10 RH 2차 클램프 풀림 [SOL]
AND NOT   T0265	// W10 RH 2차 클램프 풀림완료
OR LOAD
LOAD NOT  T0245	// W10 RH 2차 클램프 잠김완료
AND NOT   T0265	// W10 RH 2차 클램프 풀림완료
OR LOAD
LOAD      T0285	// W10 RH 2차 클램프 이상
AND NOT   M00205	// W10 RH 이상해제
OR LOAD
AND NOT   M00030	// OP LINE Emergency Stop
AND NOT   M00211	// W10 RH 공압이상
AND       M00243	// W10 RH Work Robot 간섭무
TON       T0285 50	// W10 RH 2차 클램프 이상
; L216
LOAD      P0054A	// W10 RH 3차 클램프 잠김 [SOL]
AND NOT   T0246	// W10 RH 3차 클램프 잠김완료
LOAD      P0054B	// W10 RH 3차 클램프 풀림 [SOL]
AND NOT   T0266	// W10 RH 3차 클램프 풀림완료
OR LOAD
LOAD NOT  T0246	// W10 RH 3차 클램프 잠김완료
AND NOT   T0266	// W10 RH 3차 클램프 풀림완료
OR LOAD
LOAD      T0286	// W10 RH 3차 클램프 이상
AND NOT   M00205	// W10 RH 이상해제
OR LOAD
AND NOT   M00030	// OP LINE Emergency Stop
AND NOT   M00211	// W10 RH 공압이상
AND       M00243	// W10 RH Work Robot 간섭무
TON       T0286 50	// W10 RH 3차 클램프 이상

